LIN {X 0,Y 504.364,Z 1241.928,A -85,B 0,C 180,E1 24651.564,E2 24651.564} C_VEL
LIN {X 0,Y 504.744,Z 1235.291,A -85,B 0,C 180,E1 24649.268,E2 24649.268} C_VEL
LIN {X 0,Y 505.368,Z 1226.948,A -85,B 0,C 180,E1 24646.965,E2 24646.965} C_VEL
LIN {X 0,Y 506.263,Z 1217.284,A -85,B 0,C 180,E1 24644.771,E2 24644.771} C_VEL
LIN {X 0,Y 507.475,Z 1205.57,A -85,B 0,C 180,E1 24642.573,E2 24642.573} C_VEL
LIN {X 0,Y 508.891,Z 1193.016,A -85,B 0,C 180,E1 24640.585,E2 24640.585} C_VEL
LIN {X 0,Y 510.606,Z 1178.677,A -85,B 0,C 180,E1 24638.639,E2 24638.639} C_VEL
LIN {X 0,Y 512.557,Z 1162.738,A -85,B 0,C 180,E1 24636.793,E2 24636.793} C_VEL
LIN {X 0,Y 514.559,Z 1146.108,A -85,B 0,C 180,E1 24635.16,E2 24635.16} C_VEL
LIN {X 0,Y 516.658,Z 1128.097,A -85,B 0,C 180,E1 24633.644,E2 24633.644} C_VEL
LIN {X 0,Y 518.812,Z 1108.718,A -85,B 0,C 180,E1 24632.261,E2 24632.261} C_VEL
LIN {X 0,Y 520.852,Z 1088.73,A -85,B 0,C 180,E1 24631.068,E2 24631.068} C_VEL
LIN {X 0,Y 522.71,Z 1067.81,A -85,B 0,C 180,E1 24630.048,E2 24630.048} C_VEL
LIN {X 0,Y 524.415,Z 1045.644,A -85,B 0,C 180,E1 24629.185,E2 24629.185} C_VEL
LIN {X 0,Y 525.788,Z 1023.231,A -85,B 0,C 180,E1 24628.517,E2 24628.517} C_VEL
LIN {X 0,Y 526.855,Z 1000.213,A -85,B 0,C 180,E1 24628.032,E2 24628.032} C_VEL
LIN {X 0,Y 534.144,Z 792.221,A -85,B 0,C 180,E1 24624.636,E2 24624.636} C_VEL
LIN {X 0,Y 535.779,Z 746.404,A -85,B 0,C 180,E1 24623.864,E2 24623.864} C_VEL
LIN {X 0,Y 532.938,Z 733.68,A -85,B 0,C 180,E1 24623.419,E2 24623.419} C_VEL
LIN {X 0,Y 518.726,Z 705.757,A -85,B 0,C 180,E1 24621.804,E2 24621.804} C_VEL
LIN {X 0,Y 511.196,Z 684.324,A -85,B 0,C 180,E1 24619.027,E2 24619.027} C_VEL
LIN {X 0,Y 505.862,Z 669.652,A -85,B 0,C 180,E1 24617.044,E2 24617.044} C_VEL
LIN {X 0,Y 505.876,Z 669.66,A -85,B 0,C 180,E1 24613.461,E2 24613.461} C_VEL
LIN {X 0,Y 505.86,Z 669.653,A -85,B 0,C 180,E1 24609.921,E2 24609.921} C_VEL
LIN {X 0,Y 505.869,Z 669.652,A -85,B 0,C 180,E1 24606.369,E2 24606.369} C_VEL
LIN {X 0,Y 505.872,Z 669.655,A -85,B 0,C 180,E1 24602.792,E2 24602.792} C_VEL
LIN {X 0,Y 505.863,Z 669.654,A -85,B 0,C 180,E1 24599.345,E2 24599.345} C_VEL
LIN {X 0,Y 505.866,Z 669.654,A -85,B 0,C 180,E1 24595.777,E2 24595.777} C_VEL
LIN {X 0,Y 505.86,Z 669.657,A -85,B 0,C 180,E1 24592.305,E2 24592.305} C_VEL
LIN {X 0,Y 505.871,Z 669.651,A -85,B 0,C 180,E1 24588.776,E2 24588.776} C_VEL
LIN {X 0,Y 505.866,Z 669.656,A -85,B 0,C 180,E1 24588.016,E2 24588.016} C_VEL
LIN {X 0,Y 504.876,Z 669.777,A -85,B 0,C 180,E1 24587.144,E2 24587.144} C_VEL
LIN {X 0,Y 498.35,Z 670.589,A -85,B 0,C 180,E1 24584.628,E2 24584.628} C_VEL
LIN {X 0,Y 497.917,Z 670.638,A -85,B 0,C 180,E1 24584.052,E2 24584.052} C_VEL
LIN {X 0,Y 497.931,Z 670.642,A -85,B 0,C 180,E1 24580.531,E2 24580.531} C_VEL
LIN {X 0,Y 497.921,Z 670.643,A -85,B 0,C 180,E1 24576.922,E2 24576.922} C_VEL
LIN {X 0,Y 497.921,Z 670.639,A -85,B 0,C 180,E1 24573.34,E2 24573.34} C_VEL
LIN {X 0,Y 497.923,Z 670.634,A -85,B 0,C 180,E1 24569.771,E2 24569.771} C_VEL
LIN {X 0,Y 497.917,Z 670.635,A -85,B 0,C 180,E1 24566.317,E2 24566.317} C_VEL
LIN {X 0,Y 497.936,Z 670.635,A -85,B 0,C 180,E1 24562.734,E2 24562.734} C_VEL
LIN {X 0,Y 497.917,Z 670.636,A -85,B 0,C 180,E1 24559.109,E2 24559.109} C_VEL
LIN {X 0,Y 497.936,Z 670.637,A -85,B 0,C 180,E1 24555.583,E2 24555.583} C_VEL
LIN {X 0,Y 497.923,Z 670.645,A -85,B 0,C 180,E1 24551.988,E2 24551.988} C_VEL
LIN {X 0,Y 497.926,Z 670.645,A -85,B 0,C 180,E1 24548.397,E2 24548.397} C_VEL
LIN {X 0,Y 497.925,Z 670.639,A -85,B 0,C 180,E1 24544.806,E2 24544.806} C_VEL
LIN {X 0,Y 497.922,Z 670.645,A -85,B 0,C 180,E1 24541.321,E2 24541.321} C_VEL
LIN {X 0,Y 497.925,Z 670.626,A -85,B 0,C 180,E1 24537.852,E2 24537.852} C_VEL
LIN {X 0,Y 497.919,Z 670.631,A -85,B 0,C 180,E1 24534.244,E2 24534.244} C_VEL
LIN {X 0,Y 497.955,Z 670.843,A -85,B 0,C 180,E1 24533.437,E2 24533.437} C_VEL
LIN {X 0,Y 506.765,Z 692.841,A -85,B 0,C 180,E1 24530.265,E2 24530.265} C_VEL
LIN {X 0,Y 514.424,Z 713.346,A -85,B 0,C 180,E1 24527.515,E2 24527.515} C_VEL
LIN {X 0,Y 521.93,Z 735.394,A -85,B 0,C 180,E1 24524.785,E2 24524.785} C_VEL
LIN {X 0,Y 522.331,Z 737.49,A -85,B 0,C 180,E1 24524.555,E2 24524.555} C_VEL
LIN {X 0,Y 518.753,Z 774.196,A -85,B 0,C 180,E1 24521.386,E2 24521.386} C_VEL
LIN {X 0,Y 514.969,Z 815.795,A -85,B 0,C 180,E1 24517.848,E2 24517.848} C_VEL
LIN {X 0,Y 511.442,Z 859.058,A -85,B 0,C 180,E1 24514.214,E2 24514.214} C_VEL
LIN {X 0,Y 508.148,Z 905.295,A -85,B 0,C 180,E1 24510.378,E2 24510.378} C_VEL
LIN {X 0,Y 507.992,Z 908.898,A -85,B 0,C 180,E1 24510.113,E2 24510.113} C_VEL
LIN {X 0,Y 508.886,Z 919.664,A -85,B 0,C 180,E1 24509.842,E2 24509.842} C_VEL
LIN {X 0,Y 504.35,Z 1050.728,A -85,B 0,C 180,E1 24507.128,E2 24507.128} C_VEL
LIN {X 0,Y 503.904,Z 1067.841,A -85,B 0,C 180,E1 24506.613,E2 24506.613} C_VEL
LIN {X 0,Y 503.25,Z 1083.698,A -85,B 0,C 180,E1 24505.92,E2 24505.92} C_VEL
LIN {X 0,Y 502.43,Z 1099.334,A -85,B 0,C 180,E1 24505.017,E2 24505.017} C_VEL
LIN {X 0,Y 501.517,Z 1113.85,A -85,B 0,C 180,E1 24503.937,E2 24503.937} C_VEL
LIN {X 0,Y 500.596,Z 1127.537,A -85,B 0,C 180,E1 24502.668,E2 24502.668} C_VEL
LIN {X 0,Y 499.652,Z 1140.382,A -85,B 0,C 180,E1 24501.172,E2 24501.172} C_VEL
LIN {X 0,Y 498.883,Z 1150.749,A -85,B 0,C 180,E1 24499.677,E2 24499.677} C_VEL
LIN {X 0,Y 498.188,Z 1160.6,A -85,B 0,C 180,E1 24497.883,E2 24497.883} C_VEL
LIN {X 0,Y 497.736,Z 1167.748,A -85,B 0,C 180,E1 24496.215,E2 24496.215} C_VEL
LIN {X 0,Y 497.42,Z 1173.818,A -85,B 0,C 180,E1 24494.315,E2 24494.315} C_VEL
LIN {X 0,Y 497.291,Z 1177.76,A -85,B 0,C 180,E1 24492.542,E2 24492.542} C_VEL
LIN {X 0,Y 497.285,Z 1180.289,A -85,B 0,C 180,E1 24490.521,E2 24490.521} C_VEL
LIN {X 0,Y 497.431,Z 1180.907,A -85,B 0,C 180,E1 24488.671,E2 24488.671} C_VEL
LIN {X 0,Y 497.725,Z 1179.692,A -85,B 0,C 180,E1 24486.691,E2 24486.691} C_VEL
LIN {X 0,Y 498.203,Z 1176.854,A -85,B 0,C 180,E1 24484.835,E2 24484.835} C_VEL
LIN {X 0,Y 498.95,Z 1171.888,A -85,B 0,C 180,E1 24482.872,E2 24482.872} C_VEL
LIN {X 0,Y 499.852,Z 1165.769,A -85,B 0,C 180,E1 24481.146,E2 24481.146} C_VEL
LIN {X 0,Y 501.108,Z 1157.14,A -85,B 0,C 180,E1 24479.314,E2 24479.314} C_VEL
LIN {X 0,Y 502.459,Z 1147.46,A -85,B 0,C 180,E1 24477.719,E2 24477.719} C_VEL
LIN {X 0,Y 503.927,Z 1136.358,A -85,B 0,C 180,E1 24476.246,E2 24476.246} C_VEL
LIN {X 0,Y 505.458,Z 1123.633,A -85,B 0,C 180,E1 24474.893,E2 24474.893} C_VEL
LIN {X 0,Y 506.866,Z 1110.62,A -85,B 0,C 180,E1 24473.771,E2 24473.771} C_VEL
LIN {X 0,Y 508.237,Z 1095.771,A -85,B 0,C 180,E1 24472.767,E2 24472.767} C_VEL
LIN {X 0,Y 509.323,Z 1081.041,A -85,B 0,C 180,E1 24471.988,E2 24471.988} C_VEL
LIN {X 0,Y 510.261,Z 1063.639,A -85,B 0,C 180,E1 24471.307,E2 24471.307} C_VEL
LIN {X 0,Y 513.071,Z 1023.611,A -85,B 0,C 180,E1 24470.111,E2 24470.111} C_VEL
LIN {X 0,Y 519.657,Z 948.637,A -85,B 0,C 180,E1 24468.048,E2 24468.048} C_VEL
LIN {X 0,Y 521.331,Z 927.047,A -85,B 0,C 180,E1 24467.49,E2 24467.49} C_VEL
LIN {X 0,Y 528.249,Z 885.776,A -85,B 0,C 180,E1 24463.562,E2 24463.562} C_VEL
LIN {X 0,Y 536.223,Z 847.729,A -85,B 0,C 180,E1 24459.82,E2 24459.82} C_VEL
LIN {X 0,Y 545.73,Z 811.629,A -85,B 0,C 180,E1 24456.114,E2 24456.114} C_VEL
LIN {X 0,Y 554.554,Z 784.609,A -85,B 0,C 180,E1 24453.207,E2 24453.207} C_VEL
LIN {X 0,Y 556.027,Z 780.377,A -85,B 0,C 180,E1 24452.706,E2 24452.706} C_VEL
LIN {X 0,Y 555.302,Z 773.817,A -85,B 0,C 180,E1 24450.793,E2 24450.793} C_VEL
LIN {X 0,Y 554.864,Z 769.209,A -85,B 0,C 180,E1 24448.856,E2 24448.856} C_VEL
LIN {X 0,Y 554.855,Z 767.416,A -85,B 0,C 180,E1 24447.686,E2 24447.686} C_VEL
LIN {X 0,Y 555.608,Z 765.75,A -85,B 0,C 180,E1 24445.507,E2 24445.507} C_VEL
LIN {X 0,Y 555.776,Z 766.406,A -85,B 0,C 180,E1 24444.582,E2 24444.582} C_VEL
LIN {X 0,Y 556.536,Z 769.26,A -85,B 0,C 180,E1 24442.737,E2 24442.737} C_VEL
LIN {X 0,Y 557.449,Z 773.099,A -85,B 0,C 180,E1 24441.301,E2 24441.301} C_VEL
LIN {X 0,Y 547.171,Z 799.995,A -85,B 0,C 180,E1 24438.917,E2 24438.917} C_VEL
LIN {X 0,Y 539.997,Z 825.145,A -85,B 0,C 180,E1 24436.691,E2 24436.691} C_VEL
LIN {X 0,Y 536.29,Z 846.795,A -85,B 0,C 180,E1 24434.657,E2 24434.657} C_VEL
LIN {X 0,Y 535.325,Z 864.261,A -85,B 0,C 180,E1 24432.93,E2 24432.93} C_VEL
LIN {X 0,Y 536.577,Z 881.954,A -85,B 0,C 180,E1 24431.082,E2 24431.082} C_VEL
LIN {X 0,Y 540.082,Z 898.355,A -85,B 0,C 180,E1 24429.297,E2 24429.297} C_VEL
LIN {X 0,Y 545.937,Z 914.131,A -85,B 0,C 180,E1 24427.529,E2 24427.529} C_VEL
LIN {X 0,Y 553.358,Z 927.813,A -85,B 0,C 180,E1 24425.951,E2 24425.951} C_VEL
LIN {X 0,Y 553.874,Z 928.862,A -85,B 0,C 180,E1 24425.839,E2 24425.839} C_VEL
LIN {X 0,Y 543.51,Z 949.382,A -85,B 0,C 180,E1 24425.09,E2 24425.09} C_VEL
LIN {X 0,Y 530.676,Z 977.187,A -85,B 0,C 180,E1 24423.961,E2 24423.961} C_VEL
LIN {X 0,Y 521.338,Z 1002.518,A -85,B 0,C 180,E1 24422.778,E2 24422.778} C_VEL
LIN {X 0,Y 518.892,Z 1027.417,A -85,B 0,C 180,E1 24422.456,E2 24422.456} C_VEL
LIN {X 0,Y 517.522,Z 1062.325,A -85,B 0,C 180,E1 24421.831,E2 24421.831} C_VEL
LIN {X 0,Y 516.081,Z 1085.156,A -85,B 0,C 180,E1 24421.23,E2 24421.23} C_VEL
LIN {X 0,Y 514.305,Z 1107.549,A -85,B 0,C 180,E1 24420.426,E2 24420.426} C_VEL
LIN {X 0,Y 512.324,Z 1128.678,A -85,B 0,C 180,E1 24419.458,E2 24419.458} C_VEL
LIN {X 0,Y 510.136,Z 1150.077,A -85,B 0,C 180,E1 24418.25,E2 24418.25} C_VEL
LIN {X 0,Y 507.97,Z 1169.722,A -85,B 0,C 180,E1 24416.913,E2 24416.913} C_VEL
LIN {X 0,Y 505.782,Z 1188.665,A -85,B 0,C 180,E1 24415.384,E2 24415.384} C_VEL
LIN {X 0,Y 503.683,Z 1206.377,A -85,B 0,C 180,E1 24413.684,E2 24413.684} C_VEL
LIN {X 0,Y 501.781,Z 1222.458,A -85,B 0,C 180,E1 24411.876,E2 24411.876} C_VEL
LIN {X 0,Y 500.177,Z 1236.908,A -85,B 0,C 180,E1 24409.987,E2 24409.987} C_VEL
LIN {X 0,Y 498.742,Z 1250.762,A -85,B 0,C 180,E1 24407.861,E2 24407.861} C_VEL
LIN {X 0,Y 497.682,Z 1262.373,A -85,B 0,C 180,E1 24405.735,E2 24405.735} C_VEL
LIN {X 0,Y 496.884,Z 1273.169,A -85,B 0,C 180,E1 24403.379,E2 24403.379} C_VEL
LIN {X 0,Y 496.419,Z 1281.59,A -85,B 0,C 180,E1 24401.147,E2 24401.147} C_VEL
LIN {X 0,Y 496.194,Z 1288.215,A -85,B 0,C 180,E1 24398.925,E2 24398.925} C_VEL
LIN {X 0,Y 496.115,Z 1293.775,A -85,B 0,C 180,E1 24396.477,E2 24396.477} C_VEL
LIN {X 0,Y 496.133,Z 1297.446,A -85,B 0,C 180,E1 24394.159,E2 24394.159} C_VEL
LIN {X 0,Y 496.171,Z 1299.407,A -85,B 0,C 180,E1 24391.846,E2 24391.846} C_VEL
LIN {X 0,Y 496.179,Z 1299.871,A -85,B 0,C 180,E1 24389.421,E2 24389.421} C_VEL
LIN {X 0,Y 496.163,Z 1298.798,A -85,B 0,C 180,E1 24387.226,E2 24387.226} C_VEL
LIN {X 0,Y 496.121,Z 1295.944,A -85,B 0,C 180,E1 24384.795,E2 24384.795} C_VEL
LIN {X 0,Y 496.145,Z 1291.669,A -85,B 0,C 180,E1 24382.471,E2 24382.471} C_VEL
LIN {X 0,Y 496.271,Z 1285.615,A -85,B 0,C 180,E1 24380.138,E2 24380.138} C_VEL
LIN {X 0,Y 496.616,Z 1277.824,A -85,B 0,C 180,E1 24377.794,E2 24377.794} C_VEL
LIN {X 0,Y 497.2,Z 1268.724,A -85,B 0,C 180,E1 24375.558,E2 24375.558} C_VEL
LIN {X 0,Y 498.121,Z 1257.595,A -85,B 0,C 180,E1 24373.317,E2 24373.317} C_VEL
LIN {X 0,Y 499.351,Z 1245.086,A -85,B 0,C 180,E1 24371.192,E2 24371.192} C_VEL
LIN {X 0,Y 500.876,Z 1231.302,A -85,B 0,C 180,E1 24369.185,E2 24369.185} C_VEL
LIN {X 0,Y 502.803,Z 1215.123,A -85,B 0,C 180,E1 24367.182,E2 24367.182} C_VEL
LIN {X 0,Y 504.856,Z 1198.42,A -85,B 0,C 180,E1 24365.422,E2 24365.422} C_VEL
LIN {X 0,Y 507.196,Z 1179.761,A -85,B 0,C 180,E1 24363.736,E2 24363.736} C_VEL
LIN {X 0,Y 509.611,Z 1160.303,A -85,B 0,C 180,E1 24362.239,E2 24362.239} C_VEL
LIN {X 0,Y 512.103,Z 1139.839,A -85,B 0,C 180,E1 24360.909,E2 24360.909} C_VEL
LIN {X 0,Y 514.507,Z 1118.825,A -85,B 0,C 180,E1 24359.778,E2 24359.778} C_VEL
LIN {X 0,Y 516.923,Z 1096.126,A -85,B 0,C 180,E1 24358.774,E2 24358.774} C_VEL
LIN {X 0,Y 519.31,Z 1071.964,A -85,B 0,C 180,E1 24357.938,E2 24357.938} C_VEL
LIN {X 0,Y 521.333,Z 1047.272,A -85,B 0,C 180,E1 24357.297,E2 24357.297} C_VEL
LIN {X 0,Y 523.291,Z 1020.268,A -85,B 0,C 180,E1 24356.763,E2 24356.763} C_VEL
LIN {X 0,Y 526.834,Z 993.87,A -85,B 0,C 180,E1 24356.393,E2 24356.393} C_VEL
LIN {X 0,Y 528.818,Z 981.657,A -85,B 0,C 180,E1 24356.226,E2 24356.226} C_VEL
LIN {X 0,Y 537.469,Z 962.627,A -85,B 0,C 180,E1 24355.364,E2 24355.364} C_VEL
LIN {X 0,Y 551.978,Z 933.996,A -85,B 0,C 180,E1 24354.189,E2 24354.189} C_VEL
LIN {X 0,Y 554.447,Z 929.286,A -85,B 0,C 180,E1 24354.006,E2 24354.006} C_VEL
LIN {X 0,Y 545.465,Z 913.489,A -85,B 0,C 180,E1 24352.45,E2 24352.45} C_VEL
LIN {X 0,Y 538.162,Z 895.688,A -85,B 0,C 180,E1 24350.785,E2 24350.785} C_VEL
LIN {X 0,Y 533.179,Z 877.53,A -85,B 0,C 180,E1 24349.174,E2 24349.174} C_VEL
LIN {X 0,Y 529.999,Z 856.994,A -85,B 0,C 180,E1 24347.453,E2 24347.453} C_VEL
LIN {X 0,Y 529.011,Z 834.745,A -85,B 0,C 180,E1 24345.708,E2 24345.708} C_VEL
LIN {X 0,Y 530.151,Z 810.275,A -85,B 0,C 180,E1 24343.906,E2 24343.906} C_VEL
LIN {X 0,Y 534.248,Z 775.142,A -85,B 0,C 180,E1 24341.454,E2 24341.454} C_VEL
LIN {X 0,Y 537.68,Z 769.168,A -85,B 0,C 180,E1 24340.728,E2 24340.728} C_VEL
LIN {X 0,Y 542.857,Z 759.339,A -85,B 0,C 180,E1 24339.9,E2 24339.9} C_VEL
LIN {X 0,Y 545.665,Z 757.3,A -85,B 0,C 180,E1 24339.308,E2 24339.308} C_VEL
LIN {X 0,Y 549.092,Z 755.477,A -85,B 0,C 180,E1 24338.634,E2 24338.634} C_VEL
LIN {X 0,Y 538.742,Z 835.57,A -85,B 0,C 180,E1 24336.721,E2 24336.721} C_VEL
LIN {X 0,Y 530.844,Z 913.19,A -85,B 0,C 180,E1 24334.924,E2 24334.924} C_VEL
LIN {X 0,Y 525.076,Z 987.708,A -85,B 0,C 180,E1 24333.314,E2 24333.314} C_VEL
LIN {X 0,Y 522.716,Z 1023.697,A -85,B 0,C 180,E1 24332.523,E2 24332.523} C_VEL
LIN {X 0,Y 520.89,Z 1047.072,A -85,B 0,C 180,E1 24331.798,E2 24331.798} C_VEL
LIN {X 0,Y 518.661,Z 1070.49,A -85,B 0,C 180,E1 24330.851,E2 24330.851} C_VEL
LIN {X 0,Y 516.264,Z 1092.595,A -85,B 0,C 180,E1 24329.724,E2 24329.724} C_VEL
LIN {X 0,Y 513.818,Z 1112.739,A -85,B 0,C 180,E1 24328.475,E2 24328.475} C_VEL
LIN {X 0,Y 511.287,Z 1132.087,A -85,B 0,C 180,E1 24327.045,E2 24327.045} C_VEL
LIN {X 0,Y 508.747,Z 1150.526,A -85,B 0,C 180,E1 24325.432,E2 24325.432} C_VEL
LIN {X 0,Y 506.333,Z 1167.423,A -85,B 0,C 180,E1 24323.695,E2 24323.695} C_VEL
LIN {X 0,Y 504.035,Z 1183.242,A -85,B 0,C 180,E1 24321.775,E2 24321.775} C_VEL
LIN {X 0,Y 502.033,Z 1197.078,A -85,B 0,C 180,E1 24319.791,E2 24319.791} C_VEL
LIN {X 0,Y 500.215,Z 1210.203,A -85,B 0,C 180,E1 24317.568,E2 24317.568} C_VEL
LIN {X 0,Y 498.815,Z 1221.199,A -85,B 0,C 180,E1 24315.343,E2 24315.343} C_VEL
LIN {X 0,Y 497.729,Z 1230.767,A -85,B 0,C 180,E1 24313.003,E2 24313.003} C_VEL
LIN {X 0,Y 496.982,Z 1238.369,A -85,B 0,C 180,E1 24310.667,E2 24310.667} C_VEL
LIN {X 0,Y 496.49,Z 1244.569,A -85,B 0,C 180,E1 24308.221,E2 24308.221} C_VEL
LIN {X 0,Y 496.231,Z 1249.071,A -85,B 0,C 180,E1 24305.782,E2 24305.782} C_VEL
LIN {X 0,Y 496.096,Z 1251.736,A -85,B 0,C 180,E1 24303.467,E2 24303.467} C_VEL
LIN {X 0,Y 496.049,Z 1252.986,A -85,B 0,C 180,E1 24301.039,E2 24301.039} C_VEL
LIN {X 0,Y 496.034,Z 1252.746,A -85,B 0,C 180,E1 24298.729,E2 24298.729} C_VEL
LIN {X 0,Y 496.057,Z 1250.806,A -85,B 0,C 180,E1 24296.302,E2 24296.302} C_VEL
LIN {X 0,Y 496.163,Z 1247.071,A -85,B 0,C 180,E1 24293.752,E2 24293.752} C_VEL
LIN {X 0,Y 496.395,Z 1242.114,A -85,B 0,C 180,E1 24291.428,E2 24291.428} C_VEL
LIN {X 0,Y 496.825,Z 1235.048,A -85,B 0,C 180,E1 24288.978,E2 24288.978} C_VEL
LIN {X 0,Y 497.503,Z 1226.494,A -85,B 0,C 180,E1 24286.636,E2 24286.636} C_VEL
LIN {X 0,Y 498.519,Z 1216.007,A -85,B 0,C 180,E1 24284.29,E2 24284.29} C_VEL
LIN {X 0,Y 499.765,Z 1204.724,A -85,B 0,C 180,E1 24282.175,E2 24282.175} C_VEL
LIN {X 0,Y 501.347,Z 1191.247,A -85,B 0,C 180,E1 24280.059,E2 24280.059} C_VEL
LIN {X 0,Y 503.206,Z 1176.294,A -85,B 0,C 180,E1 24278.064,E2 24278.064} C_VEL
LIN {X 0,Y 505.279,Z 1159.817,A -85,B 0,C 180,E1 24276.191,E2 24276.191} C_VEL
LIN {X 0,Y 507.389,Z 1143.021,A -85,B 0,C 180,E1 24274.557,E2 24274.557} C_VEL
LIN {X 0,Y 509.666,Z 1123.886,A -85,B 0,C 180,E1 24272.988,E2 24272.988} C_VEL
LIN {X 0,Y 511.803,Z 1104.612,A -85,B 0,C 180,E1 24271.657,E2 24271.657} C_VEL
LIN {X 0,Y 513.956,Z 1083.523,A -85,B 0,C 180,E1 24270.444,E2 24270.444} C_VEL
LIN {X 0,Y 515.867,Z 1062.333,A -85,B 0,C 180,E1 24269.448,E2 24269.448} C_VEL
LIN {X 0,Y 517.522,Z 1040.269,A -85,B 0,C 180,E1 24268.627,E2 24268.627} C_VEL
LIN {X 0,Y 518.851,Z 1017.754,A -85,B 0,C 180,E1 24268.005,E2 24268.005} C_VEL
LIN {X 0,Y 519.95,Z 991.242,A -85,B 0,C 180,E1 24267.501,E2 24267.501} C_VEL
LIN {X 0,Y 527.629,Z 784.848,A -85,B 0,C 180,E1 24264.06,E2 24264.06} C_VEL
LIN {X 0,Y 529.017,Z 747.99,A -85,B 0,C 180,E1 24263.424,E2 24263.424} C_VEL
LIN {X 0,Y 526.552,Z 737.144,A -85,B 0,C 180,E1 24263.034,E2 24263.034} C_VEL
LIN {X 0,Y 510.662,Z 706.055,A -85,B 0,C 180,E1 24261.197,E2 24261.197} C_VEL
LIN {X 0,Y 503.381,Z 685.505,A -85,B 0,C 180,E1 24258.492,E2 24258.492} C_VEL
LIN {X 0,Y 497.922,Z 670.642,A -85,B 0,C 180,E1 24256.465,E2 24256.465} C_VEL
LIN {X 0,Y 497.927,Z 670.642,A -85,B 0,C 180,E1 24252.903,E2 24252.903} C_VEL
LIN {X 0,Y 497.927,Z 670.644,A -85,B 0,C 180,E1 24249.365,E2 24249.365} C_VEL
LIN {X 0,Y 497.935,Z 670.647,A -85,B 0,C 180,E1 24245.78,E2 24245.78} C_VEL
LIN {X 0,Y 497.929,Z 670.643,A -85,B 0,C 180,E1 24242.152,E2 24242.152} C_VEL
LIN {X 0,Y 497.922,Z 670.644,A -85,B 0,C 180,E1 24238.651,E2 24238.651} C_VEL
LIN {X 0,Y 497.936,Z 670.645,A -85,B 0,C 180,E1 24235.07,E2 24235.07} C_VEL
LIN {X 0,Y 497.923,Z 670.645,A -85,B 0,C 180,E1 24231.562,E2 24231.562} C_VEL
LIN {X 0,Y 497.928,Z 670.645,A -85,B 0,C 180,E1 24228.015,E2 24228.015} C_VEL
LIN {X 0,Y 497.928,Z 670.639,A -85,B 0,C 180,E1 24224.42,E2 24224.42} C_VEL
LIN {X 0,Y 497.917,Z 670.638,A -85,B 0,C 180,E1 24224.052,E2 24224.052} C_VEL
LIN {X 0,Y 496.935,Z 670.759,A -85,B 0,C 180,E1 24223.166,E2 24223.166} C_VEL
LIN {X 0,Y 490.419,Z 671.58,A -85,B 0,C 180,E1 24220.609,E2 24220.609} C_VEL
LIN {X 0,Y 489.982,Z 671.632,A -85,B 0,C 180,E1 24220.024,E2 24220.024} C_VEL
LIN {X 0,Y 489.988,Z 671.631,A -85,B 0,C 180,E1 24216.446,E2 24216.446} C_VEL
LIN {X 0,Y 489.98,Z 671.629,A -85,B 0,C 180,E1 24212.809,E2 24212.809} C_VEL
LIN {X 0,Y 489.98,Z 671.624,A -85,B 0,C 180,E1 24209.3,E2 24209.3} C_VEL
LIN {X 0,Y 489.991,Z 671.622,A -85,B 0,C 180,E1 24205.672,E2 24205.672} C_VEL
LIN {X 0,Y 489.978,Z 671.625,A -85,B 0,C 180,E1 24202.143,E2 24202.143} C_VEL
LIN {X 0,Y 489.986,Z 671.624,A -85,B 0,C 180,E1 24198.585,E2 24198.585} C_VEL
LIN {X 0,Y 489.983,Z 671.63,A -85,B 0,C 180,E1 24194.981,E2 24194.981} C_VEL
LIN {X 0,Y 489.988,Z 671.634,A -85,B 0,C 180,E1 24191.439,E2 24191.439} C_VEL
LIN {X 0,Y 489.983,Z 671.634,A -85,B 0,C 180,E1 24187.822,E2 24187.822} C_VEL
LIN {X 0,Y 489.984,Z 671.631,A -85,B 0,C 180,E1 24184.239,E2 24184.239} C_VEL
LIN {X 0,Y 489.997,Z 671.63,A -85,B 0,C 180,E1 24180.544,E2 24180.544} C_VEL
LIN {X 0,Y 489.983,Z 671.618,A -85,B 0,C 180,E1 24176.988,E2 24176.988} C_VEL
LIN {X 0,Y 490.011,Z 671.847,A -85,B 0,C 180,E1 24174.155,E2 24174.155} C_VEL
LIN {X 0,Y 498.364,Z 692.439,A -85,B 0,C 180,E1 24171.101,E2 24171.101} C_VEL
LIN {X 0,Y 506.167,Z 713.033,A -85,B 0,C 180,E1 24168.266,E2 24168.266} C_VEL
LIN {X 0,Y 513.881,Z 735.453,A -85,B 0,C 180,E1 24165.41,E2 24165.41} C_VEL
LIN {X 0,Y 515.236,Z 740.019,A -85,B 0,C 180,E1 24164.864,E2 24164.864} C_VEL
LIN {X 0,Y 511.531,Z 776.997,A -85,B 0,C 180,E1 24161.652,E2 24161.652} C_VEL
LIN {X 0,Y 507.592,Z 818.716,A -85,B 0,C 180,E1 24158.066,E2 24158.066} C_VEL
LIN {X 0,Y 503.893,Z 862.26,A -85,B 0,C 180,E1 24154.367,E2 24154.367} C_VEL
LIN {X 0,Y 500.56,Z 907.377,A -85,B 0,C 180,E1 24150.582,E2 24150.582} C_VEL
LIN {X 0,Y 500.515,Z 909.781,A -85,B 0,C 180,E1 24150.426,E2 24150.426} C_VEL
LIN {X 0,Y 501.381,Z 920.588,A -85,B 0,C 180,E1 24150.149,E2 24150.149} C_VEL
LIN {X 0,Y 496.68,Z 1050.301,A -85,B 0,C 180,E1 24147.399,E2 24147.399} C_VEL
LIN {X 0,Y 496.206,Z 1067.96,A -85,B 0,C 180,E1 24146.865,E2 24146.865} C_VEL
LIN {X 0,Y 495.524,Z 1084.054,A -85,B 0,C 180,E1 24146.155,E2 24146.155} C_VEL
LIN {X 0,Y 494.678,Z 1099.617,A -85,B 0,C 180,E1 24145.245,E2 24145.245} C_VEL
LIN {X 0,Y 493.731,Z 1114.23,A -85,B 0,C 180,E1 24144.148,E2 24144.148} C_VEL
LIN {X 0,Y 492.81,Z 1127.454,A -85,B 0,C 180,E1 24142.912,E2 24142.912} C_VEL
LIN {X 0,Y 491.942,Z 1139,A -85,B 0,C 180,E1 24141.586,E2 24141.586} C_VEL
LIN {X 0,Y 491.08,Z 1150.184,A -85,B 0,C 180,E1 24140.003,E2 24140.003} C_VEL
LIN {X 0,Y 490.414,Z 1159.187,A -85,B 0,C 180,E1 24138.423,E2 24138.423} C_VEL
LIN {X 0,Y 489.876,Z 1167.32,A -85,B 0,C 180,E1 24136.604,E2 24136.604} C_VEL
LIN {X 0,Y 489.53,Z 1173.484,A -85,B 0,C 180,E1 24134.793,E2 24134.793} C_VEL
LIN {X 0,Y 489.348,Z 1178.3,A -85,B 0,C 180,E1 24132.749,E2 24132.749} C_VEL
LIN {X 0,Y 489.332,Z 1180.969,A -85,B 0,C 180,E1 24130.836,E2 24130.836} C_VEL
LIN {X 0,Y 489.477,Z 1181.921,A -85,B 0,C 180,E1 24128.813,E2 24128.813} C_VEL
LIN {X 0,Y 489.762,Z 1181.073,A -85,B 0,C 180,E1 24126.918,E2 24126.918} C_VEL
LIN {X 0,Y 490.271,Z 1178.356,A -85,B 0,C 180,E1 24124.914,E2 24124.914} C_VEL
LIN {X 0,Y 490.992,Z 1174.008,A -85,B 0,C 180,E1 24123.035,E2 24123.035} C_VEL
LIN {X 0,Y 492.016,Z 1167.604,A -85,B 0,C 180,E1 24121.108,E2 24121.108} C_VEL
LIN {X 0,Y 493.269,Z 1159.489,A -85,B 0,C 180,E1 24119.303,E2 24119.303} C_VEL
LIN {X 0,Y 494.684,Z 1150.259,A -85,B 0,C 180,E1 24117.683,E2 24117.683} C_VEL
LIN {X 0,Y 496.323,Z 1138.65,A -85,B 0,C 180,E1 24116.072,E2 24116.072} C_VEL
LIN {X 0,Y 497.864,Z 1126.874,A -85,B 0,C 180,E1 24114.757,E2 24114.757} C_VEL
LIN {X 0,Y 499.469,Z 1112.928,A -85,B 0,C 180,E1 24113.505,E2 24113.505} C_VEL
LIN {X 0,Y 500.92,Z 1098.61,A -85,B 0,C 180,E1 24112.487,E2 24112.487} C_VEL
LIN {X 0,Y 502.179,Z 1083.506,A -85,B 0,C 180,E1 24111.642,E2 24111.642} C_VEL
LIN {X 0,Y 503.162,Z 1066.735,A -85,B 0,C 180,E1 24110.953,E2 24110.953} C_VEL
LIN {X 0,Y 505.892,Z 1029.39,A -85,B 0,C 180,E1 24109.779,E2 24109.779} C_VEL
LIN {X 0,Y 512.761,Z 955.756,A -85,B 0,C 180,E1 24107.677,E2 24107.677} C_VEL
LIN {X 0,Y 515.019,Z 928.622,A -85,B 0,C 180,E1 24106.96,E2 24106.96} C_VEL
LIN {X 0,Y 522.253,Z 887.889,A -85,B 0,C 180,E1 24103.024,E2 24103.024} C_VEL
LIN {X 0,Y 530.696,Z 850.247,A -85,B 0,C 180,E1 24099.255,E2 24099.255} C_VEL
LIN {X 0,Y 540.105,Z 816.488,A -85,B 0,C 180,E1 24095.733,E2 24095.733} C_VEL
LIN {X 0,Y 549.352,Z 789.709,A -85,B 0,C 180,E1 24092.816,E2 24092.816} C_VEL
LIN {X 0,Y 550.844,Z 785.492,A -85,B 0,C 180,E1 24092.31,E2 24092.31} C_VEL
LIN {X 0,Y 550.394,Z 779.565,A -85,B 0,C 180,E1 24090.476,E2 24090.476} C_VEL
LIN {X 0,Y 550.194,Z 775.471,A -85,B 0,C 180,E1 24088.662,E2 24088.662} C_VEL
LIN {X 0,Y 550.251,Z 773.894,A -85,B 0,C 180,E1 24087.584,E2 24087.584} C_VEL
LIN {X 0,Y 551.076,Z 772.341,A -85,B 0,C 180,E1 24085.458,E2 24085.458} C_VEL
LIN {X 0,Y 551.221,Z 773.117,A -85,B 0,C 180,E1 24084.516,E2 24084.516} C_VEL
LIN {X 0,Y 551.914,Z 775.887,A -85,B 0,C 180,E1 24082.764,E2 24082.764} C_VEL
LIN {X 0,Y 552.46,Z 778.589,A -85,B 0,C 180,E1 24081.725,E2 24081.725} C_VEL
LIN {X 0,Y 541.566,Z 805.844,A -85,B 0,C 180,E1 24079.276,E2 24079.276} C_VEL
LIN {X 0,Y 534.284,Z 830.218,A -85,B 0,C 180,E1 24077.061,E2 24077.061} C_VEL
LIN {X 0,Y 530.559,Z 850.368,A -85,B 0,C 180,E1 24075.119,E2 24075.119} C_VEL
LIN {X 0,Y 529.282,Z 869.4,A -85,B 0,C 180,E1 24073.179,E2 24073.179} C_VEL
LIN {X 0,Y 530.561,Z 887.498,A -85,B 0,C 180,E1 24071.24,E2 24071.24} C_VEL
LIN {X 0,Y 533.862,Z 903.063,A -85,B 0,C 180,E1 24069.497,E2 24069.497} C_VEL
LIN {X 0,Y 539.786,Z 919.194,A -85,B 0,C 180,E1 24067.637,E2 24067.637} C_VEL
LIN {X 0,Y 545.938,Z 931.026,A -85,B 0,C 180,E1 24066.25,E2 24066.25} C_VEL
LIN {X 0,Y 535.777,Z 951.59,A -85,B 0,C 180,E1 24065.476,E2 24065.476} C_VEL
LIN {X 0,Y 524.83,Z 974.952,A -85,B 0,C 180,E1 24064.531,E2 24064.531} C_VEL
LIN {X 0,Y 514.891,Z 1001.395,A -85,B 0,C 180,E1 24063.294,E2 24063.294} C_VEL
LIN {X 0,Y 512.272,Z 1027.243,A -85,B 0,C 180,E1 24062.958,E2 24062.958} C_VEL
LIN {X 0,Y 510.91,Z 1051.218,A -85,B 0,C 180,E1 24062.455,E2 24062.455} C_VEL
LIN {X 0,Y 509.239,Z 1078.179,A -85,B 0,C 180,E1 24061.802,E2 24061.802} C_VEL
LIN {X 0,Y 507.496,Z 1100.809,A -85,B 0,C 180,E1 24061.043,E2 24061.043} C_VEL
LIN {X 0,Y 505.536,Z 1122.381,A -85,B 0,C 180,E1 24060.112,E2 24060.112} C_VEL
LIN {X 0,Y 503.367,Z 1143.225,A -85,B 0,C 180,E1 24058.989,E2 24058.989} C_VEL
LIN {X 0,Y 501.157,Z 1162.938,A -85,B 0,C 180,E1 24057.7,E2 24057.7} C_VEL
LIN {X 0,Y 498.803,Z 1182.648,A -85,B 0,C 180,E1 24056.166,E2 24056.166} C_VEL
LIN {X 0,Y 496.617,Z 1200.724,A -85,B 0,C 180,E1 24054.502,E2 24054.502} C_VEL
LIN {X 0,Y 494.521,Z 1217.819,A -85,B 0,C 180,E1 24052.653,E2 24052.653} C_VEL
LIN {X 0,Y 492.705,Z 1233.253,A -85,B 0,C 180,E1 24050.676,E2 24050.676} C_VEL
LIN {X 0,Y 491.203,Z 1246.856,A -85,B 0,C 180,E1 24048.636,E2 24048.636} C_VEL
LIN {X 0,Y 489.996,Z 1259.291,A -85,B 0,C 180,E1 24046.445,E2 24046.445} C_VEL
LIN {X 0,Y 489.117,Z 1269.986,A -85,B 0,C 180,E1 24044.198,E2 24044.198} C_VEL
LIN {X 0,Y 488.558,Z 1278.843,A -85,B 0,C 180,E1 24041.928,E2 24041.928} C_VEL
LIN {X 0,Y 488.232,Z 1286.686,A -85,B 0,C 180,E1 24039.428,E2 24039.428} C_VEL
LIN {X 0,Y 488.136,Z 1292.402,A -85,B 0,C 180,E1 24037.058,E2 24037.058} C_VEL
LIN {X 0,Y 488.13,Z 1296.322,A -85,B 0,C 180,E1 24034.698,E2 24034.698} C_VEL
LIN {X 0,Y 488.17,Z 1298.785,A -85,B 0,C 180,E1 24032.229,E2 24032.229} C_VEL
LIN {X 0,Y 488.204,Z 1299.536,A -85,B 0,C 180,E1 24029.998,E2 24029.998} C_VEL
LIN {X 0,Y 488.169,Z 1298.744,A -85,B 0,C 180,E1 24027.651,E2 24027.651} C_VEL
LIN {X 0,Y 488.128,Z 1296.475,A -85,B 0,C 180,E1 24025.299,E2 24025.299} C_VEL
LIN {X 0,Y 488.129,Z 1292.488,A -85,B 0,C 180,E1 24022.939,E2 24022.939} C_VEL
LIN {X 0,Y 488.239,Z 1286.593,A -85,B 0,C 180,E1 24020.45,E2 24020.45} C_VEL
LIN {X 0,Y 488.572,Z 1279.108,A -85,B 0,C 180,E1 24018.031,E2 24018.031} C_VEL
LIN {X 0,Y 489.169,Z 1269.857,A -85,B 0,C 180,E1 24015.671,E2 24015.671} C_VEL
LIN {X 0,Y 490.098,Z 1259.114,A -85,B 0,C 180,E1 24013.402,E2 24013.402} C_VEL
LIN {X 0,Y 491.35,Z 1247.043,A -85,B 0,C 180,E1 24011.243,E2 24011.243} C_VEL
LIN {X 0,Y 493.006,Z 1232.741,A -85,B 0,C 180,E1 24009.085,E2 24009.085} C_VEL
LIN {X 0,Y 494.933,Z 1217.32,A -85,B 0,C 180,E1 24007.108,E2 24007.108} C_VEL
LIN {X 0,Y 497.21,Z 1200.018,A -85,B 0,C 180,E1 24005.209,E2 24005.209} C_VEL
LIN {X 0,Y 499.657,Z 1181.743,A -85,B 0,C 180,E1 24003.495,E2 24003.495} C_VEL
LIN {X 0,Y 502.296,Z 1161.907,A -85,B 0,C 180,E1 24001.913,E2 24001.913} C_VEL
LIN {X 0,Y 504.977,Z 1141.094,A -85,B 0,C 180,E1 24000.524,E2 24000.524} C_VEL
LIN {X 0,Y 507.637,Z 1119.561,A -85,B 0,C 180,E1 23999.325,E2 23999.325} C_VEL
LIN {X 0,Y 510.395,Z 1095.576,A -85,B 0,C 180,E1 23998.237,E2 23998.237} C_VEL
LIN {X 0,Y 513.002,Z 1071.055,A -85,B 0,C 180,E1 23997.372,E2 23997.372} C_VEL
LIN {X 0,Y 515.293,Z 1044.929,A -85,B 0,C 180,E1 23996.682,E2 23996.682} C_VEL
LIN {X 0,Y 517.326,Z 1019.828,A -85,B 0,C 180,E1 23996.175,E2 23996.175} C_VEL
LIN {X 0,Y 521.032,Z 993.326,A -85,B 0,C 180,E1 23995.793,E2 23995.793} C_VEL
LIN {X 0,Y 524.148,Z 975.151,A -85,B 0,C 180,E1 23995.554,E2 23995.554} C_VEL
LIN {X 0,Y 533.694,Z 955.512,A -85,B 0,C 180,E1 23994.69,E2 23994.69} C_VEL
LIN {X 0,Y 544.849,Z 933.457,A -85,B 0,C 180,E1 23993.776,E2 23993.776} C_VEL
LIN {X 0,Y 546.068,Z 931,A -85,B 0,C 180,E1 23993.676,E2 23993.676} C_VEL
LIN {X 0,Y 537.386,Z 914.874,A -85,B 0,C 180,E1 23992.085,E2 23992.085} C_VEL
LIN {X 0,Y 530.315,Z 896.626,A -85,B 0,C 180,E1 23990.373,E2 23990.373} C_VEL
LIN {X 0,Y 525.51,Z 877.608,A -85,B 0,C 180,E1 23988.681,E2 23988.681} C_VEL
LIN {X 0,Y 522.701,Z 857.001,A -85,B 0,C 180,E1 23986.949,E2 23986.949} C_VEL
LIN {X 0,Y 522.061,Z 833.291,A -85,B 0,C 180,E1 23985.079,E2 23985.079} C_VEL
LIN {X 0,Y 523.719,Z 807.291,A -85,B 0,C 180,E1 23983.17,E2 23983.17} C_VEL
LIN {X 0,Y 524.25,Z 804.145,A -85,B 0,C 180,E1 23982.911,E2 23982.911} C_VEL
LIN {X 0,Y 528.322,Z 794.484,A -85,B 0,C 180,E1 23981.908,E2 23981.908} C_VEL
LIN {X 0,Y 533.971,Z 781.731,A -85,B 0,C 180,E1 23980.903,E2 23980.903} C_VEL
LIN {X 0,Y 539.483,Z 772.496,A -85,B 0,C 180,E1 23979.906,E2 23979.906} C_VEL
LIN {X 0,Y 543.178,Z 766.2,A -85,B 0,C 180,E1 23979.362,E2 23979.362} C_VEL
LIN {X 0,Y 544.157,Z 765.715,A -85,B 0,C 180,E1 23979.153,E2 23979.153} C_VEL
LIN {X 0,Y 533.304,Z 844.029,A -85,B 0,C 180,E1 23977.238,E2 23977.238} C_VEL
LIN {X 0,Y 525.102,Z 918.826,A -85,B 0,C 180,E1 23975.459,E2 23975.459} C_VEL
LIN {X 0,Y 519.129,Z 989.306,A -85,B 0,C 180,E1 23973.885,E2 23973.885} C_VEL
LIN {X 0,Y 516.543,Z 1024.668,A -85,B 0,C 180,E1 23973.074,E2 23973.074} C_VEL
LIN {X 0,Y 514.57,Z 1047.862,A -85,B 0,C 180,E1 23972.334,E2 23972.334} C_VEL
LIN {X 0,Y 512.272,Z 1070.268,A -85,B 0,C 180,E1 23971.41,E2 23971.41} C_VEL
LIN {X 0,Y 509.852,Z 1091.172,A -85,B 0,C 180,E1 23970.338,E2 23970.338} C_VEL
LIN {X 0,Y 507.242,Z 1111.614,A -85,B 0,C 180,E1 23969.072,E2 23969.072} C_VEL
LIN {X 0,Y 504.447,Z 1131.853,A -85,B 0,C 180,E1 23967.57,E2 23967.57} C_VEL
LIN {X 0,Y 501.847,Z 1149.75,A -85,B 0,C 180,E1 23965.998,E2 23965.998} C_VEL
LIN {X 0,Y 499.264,Z 1166.786,A -85,B 0,C 180,E1 23964.24,E2 23964.24} C_VEL
LIN {X 0,Y 496.866,Z 1182.221,A -85,B 0,C 180,E1 23962.355,E2 23962.355} C_VEL
LIN {X 0,Y 494.645,Z 1196.64,A -85,B 0,C 180,E1 23960.289,E2 23960.289} C_VEL
LIN {X 0,Y 492.724,Z 1209.621,A -85,B 0,C 180,E1 23958.089,E2 23958.089} C_VEL
LIN {X 0,Y 491.188,Z 1220.813,A -85,B 0,C 180,E1 23955.83,E2 23955.83} C_VEL
LIN {X 0,Y 489.975,Z 1230.462,A -85,B 0,C 180,E1 23953.453,E2 23953.453} C_VEL
LIN {X 0,Y 489.147,Z 1238.236,A -85,B 0,C 180,E1 23951.078,E2 23951.078} C_VEL
LIN {X 0,Y 488.589,Z 1244.598,A -85,B 0,C 180,E1 23948.592,E2 23948.592} C_VEL
LIN {X 0,Y 488.284,Z 1249.232,A -85,B 0,C 180,E1 23946.113,E2 23946.113} C_VEL
LIN {X 0,Y 488.119,Z 1252.089,A -85,B 0,C 180,E1 23943.641,E2 23943.641} C_VEL
LIN {X 0,Y 488.06,Z 1253.398,A -85,B 0,C 180,E1 23941.057,E2 23941.057} C_VEL
LIN {X 0,Y 488.043,Z 1253.116,A -85,B 0,C 180,E1 23938.709,E2 23938.709} C_VEL
LIN {X 0,Y 488.063,Z 1251.244,A -85,B 0,C 180,E1 23936.359,E2 23936.359} C_VEL
LIN {X 0,Y 488.172,Z 1247.532,A -85,B 0,C 180,E1 23933.768,E2 23933.768} C_VEL
LIN {X 0,Y 488.412,Z 1242.589,A -85,B 0,C 180,E1 23931.405,E2 23931.405} C_VEL
LIN {X 0,Y 488.829,Z 1235.88,A -85,B 0,C 180,E1 23929.034,E2 23929.034} C_VEL
LIN {X 0,Y 489.515,Z 1227.438,A -85,B 0,C 180,E1 23926.655,E2 23926.655} C_VEL
LIN {X 0,Y 490.493,Z 1217.656,A -85,B 0,C 180,E1 23924.39,E2 23924.39} C_VEL
LIN {X 0,Y 491.82,Z 1205.828,A -85,B 0,C 180,E1 23922.122,E2 23922.122} C_VEL
LIN {X 0,Y 493.439,Z 1192.468,A -85,B 0,C 180,E1 23919.973,E2 23919.973} C_VEL
LIN {X 0,Y 495.407,Z 1177.135,A -85,B 0,C 180,E1 23917.884,E2 23917.884} C_VEL
LIN {X 0,Y 497.536,Z 1160.752,A -85,B 0,C 180,E1 23915.986,E2 23915.986} C_VEL
LIN {X 0,Y 499.787,Z 1143.375,A -85,B 0,C 180,E1 23914.269,E2 23914.269} C_VEL
LIN {X 0,Y 502.142,Z 1124.233,A -85,B 0,C 180,E1 23912.678,E2 23912.678} C_VEL
LIN {X 0,Y 504.346,Z 1104.962,A -85,B 0,C 180,E1 23911.329,E2 23911.329} C_VEL
LIN {X 0,Y 506.56,Z 1084.006,A -85,B 0,C 180,E1 23910.105,E2 23910.105} C_VEL
LIN {X 0,Y 508.541,Z 1062.738,A -85,B 0,C 180,E1 23909.091,E2 23909.091} C_VEL
LIN {X 0,Y 510.231,Z 1040.93,A -85,B 0,C 180,E1 23908.268,E2 23908.268} C_VEL
LIN {X 0,Y 511.616,Z 1018.365,A -85,B 0,C 180,E1 23907.63,E2 23907.63} C_VEL
LIN {X 0,Y 512.786,Z 991.425,A -85,B 0,C 180,E1 23907.106,E2 23907.106} C_VEL
LIN {X 0,Y 520.948,Z 782.107,A -85,B 0,C 180,E1 23903.551,E2 23903.551} C_VEL
LIN {X 0,Y 522.188,Z 749.349,A -85,B 0,C 180,E1 23902.975,E2 23902.975} C_VEL
LIN {X 0,Y 520.213,Z 740.745,A -85,B 0,C 180,E1 23902.658,E2 23902.658} C_VEL
LIN {X 0,Y 504.116,Z 709.471,A -85,B 0,C 180,E1 23900.787,E2 23900.787} C_VEL
LIN {X 0,Y 502.649,Z 706.502,A -85,B 0,C 180,E1 23900.593,E2 23900.593} C_VEL
LIN {X 0,Y 494.887,Z 684.827,A -85,B 0,C 180,E1 23897.689,E2 23897.689} C_VEL
LIN {X 0,Y 489.992,Z 671.636,A -85,B 0,C 180,E1 23895.831,E2 23895.831} C_VEL
LIN {X 0,Y 489.982,Z 671.63,A -85,B 0,C 180,E1 23892.203,E2 23892.203} C_VEL
LIN {X 0,Y 489.989,Z 671.636,A -85,B 0,C 180,E1 23888.642,E2 23888.642} C_VEL
LIN {X 0,Y 489.982,Z 671.635,A -85,B 0,C 180,E1 23884.991,E2 23884.991} C_VEL
LIN {X 0,Y 489.985,Z 671.63,A -85,B 0,C 180,E1 23881.461,E2 23881.461} C_VEL
LIN {X 0,Y 489.986,Z 671.63,A -85,B 0,C 180,E1 23877.861,E2 23877.861} C_VEL
LIN {X 0,Y 489.984,Z 671.633,A -85,B 0,C 180,E1 23874.217,E2 23874.217} C_VEL
LIN {X 0,Y 489.996,Z 671.633,A -85,B 0,C 180,E1 23870.504,E2 23870.504} C_VEL
LIN {X 0,Y 489.983,Z 671.633,A -85,B 0,C 180,E1 23866.968,E2 23866.968} C_VEL
LIN {X 0,Y 489.989,Z 671.623,A -85,B 0,C 180,E1 23863.333,E2 23863.333} C_VEL
LIN {X 0,Y 489.982,Z 671.632,A -85,B 0,C 180,E1 23860.024,E2 23860.024} C_VEL
LIN {X 0,Y 489,Z 671.759,A -85,B 0,C 180,E1 23859.123,E2 23859.123} C_VEL
LIN {X 0,Y 482.504,Z 672.571,A -85,B 0,C 180,E1 23856.524,E2 23856.524} C_VEL
LIN {X 0,Y 482.057,Z 672.624,A -85,B 0,C 180,E1 23855.929,E2 23855.929} C_VEL
LIN {X 0,Y 482.048,Z 672.623,A -85,B 0,C 180,E1 23852.26,E2 23852.26} C_VEL
LIN {X 0,Y 482.058,Z 672.617,A -85,B 0,C 180,E1 23848.694,E2 23848.694} C_VEL
LIN {X 0,Y 482.054,Z 672.617,A -85,B 0,C 180,E1 23845.004,E2 23845.004} C_VEL
LIN {X 0,Y 482.046,Z 672.619,A -85,B 0,C 180,E1 23841.413,E2 23841.413} C_VEL
LIN {X 0,Y 482.057,Z 672.621,A -85,B 0,C 180,E1 23837.787,E2 23837.787} C_VEL
LIN {X 0,Y 482.051,Z 672.626,A -85,B 0,C 180,E1 23834.235,E2 23834.235} C_VEL
LIN {X 0,Y 482.05,Z 672.62,A -85,B 0,C 180,E1 23830.619,E2 23830.619} C_VEL
LIN {X 0,Y 482.05,Z 672.62,A -85,B 0,C 180,E1 23826.921,E2 23826.921} C_VEL
LIN {X 0,Y 482.054,Z 672.62,A -85,B 0,C 180,E1 23823.38,E2 23823.38} C_VEL
LIN {X 0,Y 482.055,Z 672.625,A -85,B 0,C 180,E1 23819.735,E2 23819.735} C_VEL
LIN {X 0,Y 482.045,Z 672.625,A -85,B 0,C 180,E1 23816.069,E2 23816.069} C_VEL
LIN {X 0,Y 482.049,Z 672.631,A -85,B 0,C 180,E1 23814.933,E2 23814.933} C_VEL
LIN {X 0,Y 483.508,Z 676.316,A -85,B 0,C 180,E1 23814.363,E2 23814.363} C_VEL
LIN {X 0,Y 491.928,Z 697.055,A -85,B 0,C 180,E1 23811.244,E2 23811.244} C_VEL
LIN {X 0,Y 499.705,Z 717.712,A -85,B 0,C 180,E1 23808.373,E2 23808.373} C_VEL
LIN {X 0,Y 507.183,Z 739.721,A -85,B 0,C 180,E1 23805.534,E2 23805.534} C_VEL
LIN {X 0,Y 508.069,Z 743.311,A -85,B 0,C 180,E1 23805.112,E2 23805.112} C_VEL
LIN {X 0,Y 503.975,Z 782.712,A -85,B 0,C 180,E1 23801.655,E2 23801.655} C_VEL
LIN {X 0,Y 499.66,Z 827.724,A -85,B 0,C 180,E1 23797.76,E2 23797.76} C_VEL
LIN {X 0,Y 495.715,Z 873.661,A -85,B 0,C 180,E1 23793.829,E2 23793.829} C_VEL
LIN {X 0,Y 493.014,Z 910.23,A -85,B 0,C 180,E1 23790.759,E2 23790.759} C_VEL
LIN {X 0,Y 493.892,Z 921.522,A -85,B 0,C 180,E1 23790.465,E2 23790.465} C_VEL
LIN {X 0,Y 489.136,Z 1043.911,A -85,B 0,C 180,E1 23787.805,E2 23787.805} C_VEL
LIN {X 0,Y 488.638,Z 1063.737,A -85,B 0,C 180,E1 23787.27,E2 23787.27} C_VEL
LIN {X 0,Y 487.968,Z 1080.648,A -85,B 0,C 180,E1 23786.576,E2 23786.576} C_VEL
LIN {X 0,Y 487.143,Z 1096.335,A -85,B 0,C 180,E1 23785.706,E2 23785.706} C_VEL
LIN {X 0,Y 486.16,Z 1111.359,A -85,B 0,C 180,E1 23784.629,E2 23784.629} C_VEL
LIN {X 0,Y 485.185,Z 1125.295,A -85,B 0,C 180,E1 23783.373,E2 23783.373} C_VEL
LIN {X 0,Y 484.172,Z 1138.491,A -85,B 0,C 180,E1 23781.891,E2 23781.891} C_VEL
LIN {X 0,Y 483.29,Z 1149.578,A -85,B 0,C 180,E1 23780.339,E2 23780.339} C_VEL
LIN {X 0,Y 482.529,Z 1159.535,A -85,B 0,C 180,E1 23778.61,E2 23778.61} C_VEL
LIN {X 0,Y 481.961,Z 1167.806,A -85,B 0,C 180,E1 23776.761,E2 23776.761} C_VEL
LIN {X 0,Y 481.599,Z 1174.114,A -85,B 0,C 180,E1 23774.919,E2 23774.919} C_VEL
LIN {X 0,Y 481.406,Z 1178.815,A -85,B 0,C 180,E1 23772.963,E2 23772.963} C_VEL
LIN {X 0,Y 481.387,Z 1181.744,A -85,B 0,C 180,E1 23771.017,E2 23771.017} C_VEL
LIN {X 0,Y 481.505,Z 1182.896,A -85,B 0,C 180,E1 23769.08,E2 23769.08} C_VEL
LIN {X 0,Y 481.821,Z 1182.327,A -85,B 0,C 180,E1 23767.033,E2 23767.033} C_VEL
LIN {X 0,Y 482.335,Z 1179.829,A -85,B 0,C 180,E1 23764.995,E2 23764.995} C_VEL
LIN {X 0,Y 483.085,Z 1175.772,A -85,B 0,C 180,E1 23763.085,E2 23763.085} C_VEL
LIN {X 0,Y 484.099,Z 1169.809,A -85,B 0,C 180,E1 23761.184,E2 23761.184} C_VEL
LIN {X 0,Y 485.355,Z 1162.471,A -85,B 0,C 180,E1 23759.41,E2 23759.41} C_VEL
LIN {X 0,Y 486.896,Z 1152.972,A -85,B 0,C 180,E1 23757.646,E2 23757.646} C_VEL
LIN {X 0,Y 488.471,Z 1142.752,A -85,B 0,C 180,E1 23756.127,E2 23756.127} C_VEL
LIN {X 0,Y 490.341,Z 1129.503,A -85,B 0,C 180,E1 23754.559,E2 23754.559} C_VEL
LIN {X 0,Y 492.025,Z 1116.045,A -85,B 0,C 180,E1 23753.29,E2 23753.29} C_VEL
LIN {X 0,Y 493.557,Z 1102.443,A -85,B 0,C 180,E1 23752.257,E2 23752.257} C_VEL
LIN {X 0,Y 494.951,Z 1086.956,A -85,B 0,C 180,E1 23751.344,E2 23751.344} C_VEL
LIN {X 0,Y 496.064,Z 1070.675,A -85,B 0,C 180,E1 23750.618,E2 23750.618} C_VEL
LIN {X 0,Y 498.691,Z 1035.572,A -85,B 0,C 180,E1 23749.45,E2 23749.45} C_VEL
LIN {X 0,Y 506.039,Z 961.807,A -85,B 0,C 180,E1 23747.261,E2 23747.261} C_VEL
LIN {X 0,Y 508.879,Z 930.354,A -85,B 0,C 180,E1 23746.405,E2 23746.405} C_VEL
LIN {X 0,Y 515.809,Z 892.887,A -85,B 0,C 180,E1 23742.747,E2 23742.747} C_VEL
LIN {X 0,Y 524.292,Z 856.411,A -85,B 0,C 180,E1 23739.048,E2 23739.048} C_VEL
LIN {X 0,Y 534.212,Z 822.336,A -85,B 0,C 180,E1 23735.448,E2 23735.448} C_VEL
LIN {X 0,Y 544.197,Z 794.857,A -85,B 0,C 180,E1 23732.418,E2 23732.418} C_VEL
LIN {X 0,Y 545.803,Z 790.745,A -85,B 0,C 180,E1 23731.913,E2 23731.913} C_VEL
LIN {X 0,Y 545.524,Z 785.166,A -85,B 0,C 180,E1 23730.096,E2 23730.096} C_VEL
LIN {X 0,Y 545.538,Z 781.595,A -85,B 0,C 180,E1 23728.386,E2 23728.386} C_VEL
LIN {X 0,Y 545.664,Z 780.156,A -85,B 0,C 180,E1 23727.251,E2 23727.251} C_VEL
LIN {X 0,Y 546.549,Z 778.935,A -85,B 0,C 180,E1 23725.408,E2 23725.408} C_VEL
LIN {X 0,Y 546.702,Z 780.204,A -85,B 0,C 180,E1 23724.178,E2 23724.178} C_VEL
LIN {X 0,Y 547.288,Z 782.485,A -85,B 0,C 180,E1 23722.8,E2 23722.8} C_VEL
LIN {X 0,Y 547.557,Z 784.121,A -85,B 0,C 180,E1 23722.162,E2 23722.162} C_VEL
LIN {X 0,Y 536.082,Z 811.403,A -85,B 0,C 180,E1 23719.668,E2 23719.668} C_VEL
LIN {X 0,Y 528.965,Z 834.107,A -85,B 0,C 180,E1 23717.559,E2 23717.559} C_VEL
LIN {X 0,Y 524.725,Z 855.419,A -85,B 0,C 180,E1 23715.45,E2 23715.45} C_VEL
LIN {X 0,Y 523.335,Z 873.067,A -85,B 0,C 180,E1 23713.604,E2 23713.604} C_VEL
LIN {X 0,Y 524.335,Z 891.469,A -85,B 0,C 180,E1 23711.574,E2 23711.574} C_VEL
LIN {X 0,Y 527.672,Z 907.787,A -85,B 0,C 180,E1 23709.706,E2 23709.706} C_VEL
LIN {X 0,Y 533.253,Z 923.34,A -85,B 0,C 180,E1 23707.869,E2 23707.869} C_VEL
LIN {X 0,Y 538.17,Z 933.25,A -85,B 0,C 180,E1 23706.683,E2 23706.683} C_VEL
LIN {X 0,Y 519.32,Z 972.34,A -85,B 0,C 180,E1 23705.145,E2 23705.145} C_VEL
LIN {X 0,Y 509.067,Z 998.406,A -85,B 0,C 180,E1 23703.903,E2 23703.903} C_VEL
LIN {X 0,Y 508.485,Z 1000.854,A -85,B 0,C 180,E1 23703.828,E2 23703.828} C_VEL
LIN {X 0,Y 505.727,Z 1027.324,A -85,B 0,C 180,E1 23703.476,E2 23703.476} C_VEL
LIN {X 0,Y 504.12,Z 1052.636,A -85,B 0,C 180,E1 23702.917,E2 23702.917} C_VEL
LIN {X 0,Y 501.019,Z 1090.242,A -85,B 0,C 180,E1 23701.787,E2 23701.787} C_VEL
LIN {X 0,Y 499.075,Z 1112.286,A -85,B 0,C 180,E1 23700.921,E2 23700.921} C_VEL
LIN {X 0,Y 496.958,Z 1133.246,A -85,B 0,C 180,E1 23699.889,E2 23699.889} C_VEL
LIN {X 0,Y 494.621,Z 1154.026,A -85,B 0,C 180,E1 23698.624,E2 23698.624} C_VEL
LIN {X 0,Y 492.369,Z 1172.844,A -85,B 0,C 180,E1 23697.252,E2 23697.252} C_VEL
LIN {X 0,Y 490.008,Z 1191.704,A -85,B 0,C 180,E1 23695.63,E2 23695.63} C_VEL
LIN {X 0,Y 487.837,Z 1209.04,A -85,B 0,C 180,E1 23693.877,E2 23693.877} C_VEL
LIN {X 0,Y 485.793,Z 1225.327,A -85,B 0,C 180,E1 23691.934,E2 23691.934} C_VEL
LIN {X 0,Y 484.085,Z 1239.64,A -85,B 0,C 180,E1 23689.924,E2 23689.924} C_VEL
LIN {X 0,Y 482.589,Z 1253.581,A -85,B 0,C 180,E1 23687.619,E2 23687.619} C_VEL
LIN {X 0,Y 481.533,Z 1264.833,A -85,B 0,C 180,E1 23685.412,E2 23685.412} C_VEL
LIN {X 0,Y 480.814,Z 1274.617,A -85,B 0,C 180,E1 23683.099,E2 23683.099} C_VEL
LIN {X 0,Y 480.359,Z 1282.746,A -85,B 0,C 180,E1 23680.736,E2 23680.736} C_VEL
LIN {X 0,Y 480.177,Z 1289.198,A -85,B 0,C 180,E1 23678.38,E2 23678.38} C_VEL
LIN {X 0,Y 480.131,Z 1293.831,A -85,B 0,C 180,E1 23676.095,E2 23676.095} C_VEL
LIN {X 0,Y 480.158,Z 1297.253,A -85,B 0,C 180,E1 23673.58,E2 23673.58} C_VEL
LIN {X 0,Y 480.2,Z 1298.945,A -85,B 0,C 180,E1 23671.191,E2 23671.191} C_VEL
LIN {X 0,Y 480.199,Z 1298.931,A -85,B 0,C 180,E1 23668.805,E2 23668.805} C_VEL
LIN {X 0,Y 480.15,Z 1297.3,A -85,B 0,C 180,E1 23666.297,E2 23666.297} C_VEL
LIN {X 0,Y 480.123,Z 1294.316,A -85,B 0,C 180,E1 23664.022,E2 23664.022} C_VEL
LIN {X 0,Y 480.176,Z 1289.39,A -85,B 0,C 180,E1 23661.539,E2 23661.539} C_VEL
LIN {X 0,Y 480.385,Z 1282.817,A -85,B 0,C 180,E1 23659.08,E2 23659.08} C_VEL
LIN {X 0,Y 480.883,Z 1274.587,A -85,B 0,C 180,E1 23656.683,E2 23656.683} C_VEL
LIN {X 0,Y 481.68,Z 1264.723,A -85,B 0,C 180,E1 23654.343,E2 23654.343} C_VEL
LIN {X 0,Y 482.873,Z 1253.047,A -85,B 0,C 180,E1 23652.028,E2 23652.028} C_VEL
LIN {X 0,Y 484.425,Z 1239.949,A -85,B 0,C 180,E1 23649.835,E2 23649.835} C_VEL
LIN {X 0,Y 486.299,Z 1225.36,A -85,B 0,C 180,E1 23647.769,E2 23647.769} C_VEL
LIN {X 0,Y 488.636,Z 1208.366,A -85,B 0,C 180,E1 23645.712,E2 23645.712} C_VEL
LIN {X 0,Y 491.189,Z 1190.401,A -85,B 0,C 180,E1 23643.861,E2 23643.861} C_VEL
LIN {X 0,Y 493.916,Z 1171.292,A -85,B 0,C 180,E1 23642.183,E2 23642.183} C_VEL
LIN {X 0,Y 496.811,Z 1150.622,A -85,B 0,C 180,E1 23640.653,E2 23640.653} C_VEL
LIN {X 0,Y 499.711,Z 1129.034,A -85,B 0,C 180,E1 23639.319,E2 23639.319} C_VEL
LIN {X 0,Y 502.592,Z 1106.705,A -85,B 0,C 180,E1 23638.182,E2 23638.182} C_VEL
LIN {X 0,Y 505.487,Z 1082.225,A -85,B 0,C 180,E1 23637.179,E2 23637.179} C_VEL
LIN {X 0,Y 508.225,Z 1056.68,A -85,B 0,C 180,E1 23636.386,E2 23636.386} C_VEL
LIN {X 0,Y 510.933,Z 1024.635,A -85,B 0,C 180,E1 23635.65,E2 23635.65} C_VEL
LIN {X 0,Y 514.827,Z 996.352,A -85,B 0,C 180,E1 23635.208,E2 23635.208} C_VEL
LIN {X 0,Y 519.537,Z 969.212,A -85,B 0,C 180,E1 23634.88,E2 23634.88} C_VEL
LIN {X 0,Y 537.73,Z 932.636,A -85,B 0,C 180,E1 23633.336,E2 23633.336} C_VEL
LIN {X 0,Y 529.347,Z 916.206,A -85,B 0,C 180,E1 23631.715,E2 23631.715} C_VEL
LIN {X 0,Y 522.658,Z 898.007,A -85,B 0,C 180,E1 23629.998,E2 23629.998} C_VEL
LIN {X 0,Y 518.027,Z 878.41,A -85,B 0,C 180,E1 23628.246,E2 23628.246} C_VEL
LIN {X 0,Y 515.497,Z 857.573,A -85,B 0,C 180,E1 23626.481,E2 23626.481} C_VEL
LIN {X 0,Y 515.175,Z 835.423,A -85,B 0,C 180,E1 23624.695,E2 23624.695} C_VEL
LIN {X 0,Y 518.021,Z 825.712,A -85,B 0,C 180,E1 23623.627,E2 23623.627} C_VEL
LIN {X 0,Y 522.541,Z 812.796,A -85,B 0,C 180,E1 23622.525,E2 23622.525} C_VEL
LIN {X 0,Y 524.019,Z 809.062,A -85,B 0,C 180,E1 23622.208,E2 23622.208} C_VEL
LIN {X 0,Y 528.795,Z 798.967,A -85,B 0,C 180,E1 23621.185,E2 23621.185} C_VEL
LIN {X 0,Y 535.113,Z 786.094,A -85,B 0,C 180,E1 23620.159,E2 23620.159} C_VEL
LIN {X 0,Y 538.572,Z 781.035,A -85,B 0,C 180,E1 23619.558,E2 23619.558} C_VEL
LIN {X 0,Y 527.139,Z 859.43,A -85,B 0,C 180,E1 23617.603,E2 23617.603} C_VEL
LIN {X 0,Y 518.849,Z 931.026,A -85,B 0,C 180,E1 23615.863,E2 23615.863} C_VEL
LIN {X 0,Y 512.679,Z 999.044,A -85,B 0,C 180,E1 23614.3,E2 23614.3} C_VEL
LIN {X 0,Y 510.303,Z 1028.403,A -85,B 0,C 180,E1 23613.572,E2 23613.572} C_VEL
LIN {X 0,Y 508.125,Z 1051.214,A -85,B 0,C 180,E1 23612.799,E2 23612.799} C_VEL
LIN {X 0,Y 505.708,Z 1072.946,A -85,B 0,C 180,E1 23611.865,E2 23611.865} C_VEL
LIN {X 0,Y 502.906,Z 1095.399,A -85,B 0,C 180,E1 23610.663,E2 23610.663} C_VEL
LIN {X 0,Y 500.07,Z 1115.817,A -85,B 0,C 180,E1 23609.332,E2 23609.332} C_VEL
LIN {X 0,Y 497.156,Z 1135.333,A -85,B 0,C 180,E1 23607.814,E2 23607.814} C_VEL
LIN {X 0,Y 494.34,Z 1153.27,A -85,B 0,C 180,E1 23606.164,E2 23606.164} C_VEL
LIN {X 0,Y 491.659,Z 1169.793,A -85,B 0,C 180,E1 23604.384,E2 23604.384} C_VEL
LIN {X 0,Y 489.193,Z 1184.954,A -85,B 0,C 180,E1 23602.471,E2 23602.471} C_VEL
LIN {X 0,Y 486.825,Z 1199.39,A -85,B 0,C 180,E1 23600.311,E2 23600.311} C_VEL
LIN {X 0,Y 484.888,Z 1211.617,A -85,B 0,C 180,E1 23598.142,E2 23598.142} C_VEL
LIN {X 0,Y 483.217,Z 1223.015,A -85,B 0,C 180,E1 23595.728,E2 23595.728} C_VEL
LIN {X 0,Y 482.018,Z 1232.204,A -85,B 0,C 180,E1 23593.37,E2 23593.37} C_VEL
LIN {X 0,Y 481.152,Z 1239.869,A -85,B 0,C 180,E1 23590.901,E2 23590.901} C_VEL
LIN {X 0,Y 480.609,Z 1245.64,A -85,B 0,C 180,E1 23588.494,E2 23588.494} C_VEL
LIN {X 0,Y 480.306,Z 1249.898,A -85,B 0,C 180,E1 23586.095,E2 23586.095} C_VEL
LIN {X 0,Y 480.138,Z 1252.559,A -85,B 0,C 180,E1 23583.701,E2 23583.701} C_VEL
LIN {X 0,Y 480.07,Z 1253.797,A -85,B 0,C 180,E1 23581.193,E2 23581.193} C_VEL
LIN {X 0,Y 480.054,Z 1253.534,A -85,B 0,C 180,E1 23578.807,E2 23578.807} C_VEL
LIN {X 0,Y 480.071,Z 1251.68,A -85,B 0,C 180,E1 23576.418,E2 23576.418} C_VEL
LIN {X 0,Y 480.175,Z 1248.202,A -85,B 0,C 180,E1 23573.904,E2 23573.904} C_VEL
LIN {X 0,Y 480.409,Z 1243.312,A -85,B 0,C 180,E1 23571.502,E2 23571.502} C_VEL
LIN {X 0,Y 480.831,Z 1236.698,A -85,B 0,C 180,E1 23569.092,E2 23569.092} C_VEL
LIN {X 0,Y 481.57,Z 1227.883,A -85,B 0,C 180,E1 23566.553,E2 23566.553} C_VEL
LIN {X 0,Y 482.582,Z 1218.086,A -85,B 0,C 180,E1 23564.251,E2 23564.251} C_VEL
LIN {X 0,Y 483.957,Z 1206.235,A -85,B 0,C 180,E1 23561.946,E2 23561.946} C_VEL
LIN {X 0,Y 485.633,Z 1192.859,A -85,B 0,C 180,E1 23559.763,E2 23559.763} C_VEL
LIN {X 0,Y 487.603,Z 1178.019,A -85,B 0,C 180,E1 23557.705,E2 23557.705} C_VEL
LIN {X 0,Y 489.722,Z 1162.23,A -85,B 0,C 180,E1 23555.835,E2 23555.835} C_VEL
LIN {X 0,Y 492.11,Z 1144.322,A -85,B 0,C 180,E1 23554.032,E2 23554.032} C_VEL
LIN {X 0,Y 494.528,Z 1125.241,A -85,B 0,C 180,E1 23552.418,E2 23552.418} C_VEL
LIN {X 0,Y 496.797,Z 1106.085,A -85,B 0,C 180,E1 23551.05,E2 23551.05} C_VEL
LIN {X 0,Y 499.067,Z 1085.299,A -85,B 0,C 180,E1 23549.809,E2 23549.809} C_VEL
LIN {X 0,Y 501.105,Z 1064.318,A -85,B 0,C 180,E1 23548.782,E2 23548.782} C_VEL
LIN {X 0,Y 502.936,Z 1041.456,A -85,B 0,C 180,E1 23547.901,E2 23547.901} C_VEL
LIN {X 0,Y 504.366,Z 1018.959,A -85,B 0,C 180,E1 23547.253,E2 23547.253} C_VEL
LIN {X 0,Y 505.572,Z 992.417,A -85,B 0,C 180,E1 23546.724,E2 23546.724} C_VEL
LIN {X 0,Y 514.074,Z 784.251,A -85,B 0,C 180,E1 23543.116,E2 23543.116} C_VEL
LIN {X 0,Y 515.433,Z 750.903,A -85,B 0,C 180,E1 23542.519,E2 23542.519} C_VEL
LIN {X 0,Y 513.827,Z 744.191,A -85,B 0,C 180,E1 23542.261,E2 23542.261} C_VEL
LIN {X 0,Y 496.759,Z 710.979,A -85,B 0,C 180,E1 23540.234,E2 23540.234} C_VEL
LIN {X 0,Y 494.51,Z 706.689,A -85,B 0,C 180,E1 23539.937,E2 23539.937} C_VEL
LIN {X 0,Y 486.912,Z 685.592,A -85,B 0,C 180,E1 23537.063,E2 23537.063} C_VEL
LIN {X 0,Y 482.055,Z 672.619,A -85,B 0,C 180,E1 23535.215,E2 23535.215} C_VEL
LIN {X 0,Y 482.056,Z 672.623,A -85,B 0,C 180,E1 23531.588,E2 23531.588} C_VEL
LIN {X 0,Y 482.051,Z 672.622,A -85,B 0,C 180,E1 23527.981,E2 23527.981} C_VEL
LIN {X 0,Y 482.049,Z 672.616,A -85,B 0,C 180,E1 23524.348,E2 23524.348} C_VEL
LIN {X 0,Y 482.056,Z 672.612,A -85,B 0,C 180,E1 23520.821,E2 23520.821} C_VEL
LIN {X 0,Y 482.054,Z 672.625,A -85,B 0,C 180,E1 23517.146,E2 23517.146} C_VEL
LIN {X 0,Y 482.058,Z 672.622,A -85,B 0,C 180,E1 23513.536,E2 23513.536} C_VEL
LIN {X 0,Y 482.057,Z 672.62,A -85,B 0,C 180,E1 23509.889,E2 23509.889} C_VEL
LIN {X 0,Y 482.043,Z 672.624,A -85,B 0,C 180,E1 23506.263,E2 23506.263} C_VEL
LIN {X 0,Y 482.058,Z 672.61,A -85,B 0,C 180,E1 23502.703,E2 23502.703} C_VEL
LIN {X 0,Y 482.041,Z 672.612,A -85,B 0,C 180,E1 23499.072,E2 23499.072} C_VEL
LIN {X 0,Y 482.057,Z 672.624,A -85,B 0,C 180,E1 23495.929,E2 23495.929} C_VEL
LIN {X 0,Y 481.057,Z 672.745,A -85,B 0,C 180,E1 23495.013,E2 23495.013} C_VEL
LIN {X 0,Y 474.551,Z 673.559,A -85,B 0,C 180,E1 23492.372,E2 23492.372} C_VEL
LIN {X 0,Y 474.105,Z 673.611,A -85,B 0,C 180,E1 23491.767,E2 23491.767} C_VEL
LIN {X 0,Y 474.115,Z 673.611,A -85,B 0,C 180,E1 23488.189,E2 23488.189} C_VEL
LIN {X 0,Y 474.103,Z 673.611,A -85,B 0,C 180,E1 23484.434,E2 23484.434} C_VEL
LIN {X 0,Y 474.105,Z 673.611,A -85,B 0,C 180,E1 23480.901,E2 23480.901} C_VEL
LIN {X 0,Y 474.105,Z 673.612,A -85,B 0,C 180,E1 23477.208,E2 23477.208} C_VEL
LIN {X 0,Y 474.105,Z 673.611,A -85,B 0,C 180,E1 23473.659,E2 23473.659} C_VEL
LIN {X 0,Y 474.109,Z 673.605,A -85,B 0,C 180,E1 23470.024,E2 23470.024} C_VEL
LIN {X 0,Y 474.106,Z 673.612,A -85,B 0,C 180,E1 23466.38,E2 23466.38} C_VEL
LIN {X 0,Y 474.112,Z 673.606,A -85,B 0,C 180,E1 23462.767,E2 23462.767} C_VEL
LIN {X 0,Y 474.108,Z 673.612,A -85,B 0,C 180,E1 23459.133,E2 23459.133} C_VEL
LIN {X 0,Y 474.136,Z 673.807,A -85,B 0,C 180,E1 23455.684,E2 23455.684} C_VEL
LIN {X 0,Y 483.221,Z 695.928,A -85,B 0,C 180,E1 23452.233,E2 23452.233} C_VEL
LIN {X 0,Y 490.96,Z 716.135,A -85,B 0,C 180,E1 23449.332,E2 23449.332} C_VEL
LIN {X 0,Y 498.479,Z 737.808,A -85,B 0,C 180,E1 23446.45,E2 23446.45} C_VEL
LIN {X 0,Y 501.006,Z 745.865,A -85,B 0,C 180,E1 23445.438,E2 23445.438} C_VEL
LIN {X 0,Y 496.638,Z 786.335,A -85,B 0,C 180,E1 23441.851,E2 23441.851} C_VEL
LIN {X 0,Y 492.162,Z 831.237,A -85,B 0,C 180,E1 23437.921,E2 23437.921} C_VEL
LIN {X 0,Y 488.15,Z 876.554,A -85,B 0,C 180,E1 23434,E2 23434} C_VEL
LIN {X 0,Y 485.542,Z 910.886,A -85,B 0,C 180,E1 23431.095,E2 23431.095} C_VEL
LIN {X 0,Y 486.413,Z 922.266,A -85,B 0,C 180,E1 23430.792,E2 23430.792} C_VEL
LIN {X 0,Y 481.377,Z 1047.188,A -85,B 0,C 180,E1 23427.995,E2 23427.995} C_VEL
LIN {X 0,Y 480.879,Z 1065.603,A -85,B 0,C 180,E1 23427.466,E2 23427.466} C_VEL
LIN {X 0,Y 480.158,Z 1082.786,A -85,B 0,C 180,E1 23426.731,E2 23426.731} C_VEL
LIN {X 0,Y 479.306,Z 1098.079,A -85,B 0,C 180,E1 23425.849,E2 23425.849} C_VEL
LIN {X 0,Y 478.274,Z 1113.391,A -85,B 0,C 180,E1 23424.716,E2 23424.716} C_VEL
LIN {X 0,Y 477.26,Z 1127.215,A -85,B 0,C 180,E1 23423.423,E2 23423.423} C_VEL
LIN {X 0,Y 476.25,Z 1140.011,A -85,B 0,C 180,E1 23421.945,E2 23421.945} C_VEL
LIN {X 0,Y 475.32,Z 1151.333,A -85,B 0,C 180,E1 23420.31,E2 23420.31} C_VEL
LIN {X 0,Y 474.556,Z 1161.114,A -85,B 0,C 180,E1 23418.552,E2 23418.552} C_VEL
LIN {X 0,Y 473.988,Z 1169.248,A -85,B 0,C 180,E1 23416.672,E2 23416.672} C_VEL
LIN {X 0,Y 473.626,Z 1175.436,A -85,B 0,C 180,E1 23414.792,E2 23414.792} C_VEL
LIN {X 0,Y 473.446,Z 1180.302,A -85,B 0,C 180,E1 23412.664,E2 23412.664} C_VEL
LIN {X 0,Y 473.445,Z 1182.96,A -85,B 0,C 180,E1 23410.711,E2 23410.711} C_VEL
LIN {X 0,Y 473.63,Z 1183.96,A -85,B 0,C 180,E1 23408.621,E2 23408.621} C_VEL
LIN {X 0,Y 473.969,Z 1183.164,A -85,B 0,C 180,E1 23406.663,E2 23406.663} C_VEL
LIN {X 0,Y 474.571,Z 1180.506,A -85,B 0,C 180,E1 23404.592,E2 23404.592} C_VEL
LIN {X 0,Y 475.423,Z 1176.144,A -85,B 0,C 180,E1 23402.619,E2 23402.619} C_VEL
LIN {X 0,Y 476.62,Z 1169.725,A -85,B 0,C 180,E1 23400.601,E2 23400.601} C_VEL
LIN {X 0,Y 478.11,Z 1161.395,A -85,B 0,C 180,E1 23398.682,E2 23398.682} C_VEL
LIN {X 0,Y 479.708,Z 1152.125,A -85,B 0,C 180,E1 23397.013,E2 23397.013} C_VEL
LIN {X 0,Y 481.578,Z 1140.603,A -85,B 0,C 180,E1 23395.355,E2 23395.355} C_VEL
LIN {X 0,Y 483.383,Z 1128.308,A -85,B 0,C 180,E1 23393.944,E2 23393.944} C_VEL
LIN {X 0,Y 485.125,Z 1115.141,A -85,B 0,C 180,E1 23392.718,E2 23392.718} C_VEL
LIN {X 0,Y 486.835,Z 1100.103,A -85,B 0,C 180,E1 23391.615,E2 23391.615} C_VEL
LIN {X 0,Y 488.247,Z 1085.107,A -85,B 0,C 180,E1 23390.749,E2 23390.749} C_VEL
LIN {X 0,Y 489.439,Z 1068.059,A -85,B 0,C 180,E1 23390.015,E2 23390.015} C_VEL
LIN {X 0,Y 492.679,Z 1030.711,A -85,B 0,C 180,E1 23388.754,E2 23388.754} C_VEL
LIN {X 0,Y 499.562,Z 965.705,A -85,B 0,C 180,E1 23386.773,E2 23386.773} C_VEL
LIN {X 0,Y 502.806,Z 932.185,A -85,B 0,C 180,E1 23385.842,E2 23385.842} C_VEL
LIN {X 0,Y 502.958,Z 930.038,A -85,B 0,C 180,E1 23385.67,E2 23385.67} C_VEL
LIN {X 0,Y 511.171,Z 889.858,A -85,B 0,C 180,E1 23381.643,E2 23381.643} C_VEL
LIN {X 0,Y 520.345,Z 854.077,A -85,B 0,C 180,E1 23377.934,E2 23377.934} C_VEL
LIN {X 0,Y 531.007,Z 820.785,A -85,B 0,C 180,E1 23374.336,E2 23374.336} C_VEL
LIN {X 0,Y 540.786,Z 796.114,A -85,B 0,C 180,E1 23371.538,E2 23371.538} C_VEL
LIN {X 0,Y 540.789,Z 790.768,A -85,B 0,C 180,E1 23369.684,E2 23369.684} C_VEL
LIN {X 0,Y 541.037,Z 787.258,A -85,B 0,C 180,E1 23367.821,E2 23367.821} C_VEL
LIN {X 0,Y 541.971,Z 785.498,A -85,B 0,C 180,E1 23365.501,E2 23365.501} C_VEL
LIN {X 0,Y 542.099,Z 786.426,A -85,B 0,C 180,E1 23364.478,E2 23364.478} C_VEL
LIN {X 0,Y 542.625,Z 788.876,A -85,B 0,C 180,E1 23362.925,E2 23362.925} C_VEL
LIN {X 0,Y 542.735,Z 789.681,A -85,B 0,C 180,E1 23362.609,E2 23362.609} C_VEL
LIN {X 0,Y 530.715,Z 817.105,A -85,B 0,C 180,E1 23360.064,E2 23360.064} C_VEL
LIN {X 0,Y 523.324,Z 839.611,A -85,B 0,C 180,E1 23357.915,E2 23357.915} C_VEL
LIN {X 0,Y 519.032,Z 859.867,A -85,B 0,C 180,E1 23355.854,E2 23355.854} C_VEL
LIN {X 0,Y 517.419,Z 878.233,A -85,B 0,C 180,E1 23353.879,E2 23353.879} C_VEL
LIN {X 0,Y 518.202,Z 895.443,A -85,B 0,C 180,E1 23351.932,E2 23351.932} C_VEL
LIN {X 0,Y 521.352,Z 912.027,A -85,B 0,C 180,E1 23349.975,E2 23349.975} C_VEL
LIN {X 0,Y 527.163,Z 928.453,A -85,B 0,C 180,E1 23347.992,E2 23347.992} C_VEL
LIN {X 0,Y 530.472,Z 935.528,A -85,B 0,C 180,E1 23347.125,E2 23347.125} C_VEL
LIN {X 0,Y 512.762,Z 972.302,A -85,B 0,C 180,E1 23345.663,E2 23345.663} C_VEL
LIN {X 0,Y 502.349,Z 999.002,A -85,B 0,C 180,E1 23344.402,E2 23344.402} C_VEL
LIN {X 0,Y 499.28,Z 1027.08,A -85,B 0,C 180,E1 23344.018,E2 23344.018} C_VEL
LIN {X 0,Y 497.514,Z 1052.973,A -85,B 0,C 180,E1 23343.433,E2 23343.433} C_VEL
LIN {X 0,Y 495.266,Z 1075.906,A -85,B 0,C 180,E1 23342.719,E2 23342.719} C_VEL
LIN {X 0,Y 491.861,Z 1110.571,A -85,B 0,C 180,E1 23341.358,E2 23341.358} C_VEL
LIN {X 0,Y 489.612,Z 1132.129,A -85,B 0,C 180,E1 23340.291,E2 23340.291} C_VEL
LIN {X 0,Y 487.205,Z 1152.964,A -85,B 0,C 180,E1 23339.014,E2 23339.014} C_VEL
LIN {X 0,Y 484.799,Z 1172.432,A -85,B 0,C 180,E1 23337.58,E2 23337.58} C_VEL
LIN {X 0,Y 482.363,Z 1191.309,A -85,B 0,C 180,E1 23335.935,E2 23335.935} C_VEL
LIN {X 0,Y 480.174,Z 1208.213,A -85,B 0,C 180,E1 23334.206,E2 23334.206} C_VEL
LIN {X 0,Y 478.054,Z 1224.48,A -85,B 0,C 180,E1 23332.243,E2 23332.243} C_VEL
LIN {X 0,Y 476.291,Z 1238.817,A -85,B 0,C 180,E1 23330.215,E2 23330.215} C_VEL
LIN {X 0,Y 474.736,Z 1252.677,A -85,B 0,C 180,E1 23327.907,E2 23327.907} C_VEL
LIN {X 0,Y 473.632,Z 1263.999,A -85,B 0,C 180,E1 23325.676,E2 23325.676} C_VEL
LIN {X 0,Y 472.864,Z 1273.855,A -85,B 0,C 180,E1 23323.324,E2 23323.324} C_VEL
LIN {X 0,Y 472.374,Z 1282.279,A -85,B 0,C 180,E1 23320.857,E2 23320.857} C_VEL
LIN {X 0,Y 472.182,Z 1288.899,A -85,B 0,C 180,E1 23318.4,E2 23318.4} C_VEL
LIN {X 0,Y 472.137,Z 1293.521,A -85,B 0,C 180,E1 23316.077,E2 23316.077} C_VEL
LIN {X 0,Y 472.17,Z 1296.907,A -85,B 0,C 180,E1 23313.519,E2 23313.519} C_VEL
LIN {X 0,Y 472.211,Z 1298.564,A -85,B 0,C 180,E1 23311.09,E2 23311.09} C_VEL
LIN {X 0,Y 472.207,Z 1298.503,A -85,B 0,C 180,E1 23308.664,E2 23308.664} C_VEL
LIN {X 0,Y 472.152,Z 1296.813,A -85,B 0,C 180,E1 23306.113,E2 23306.113} C_VEL
LIN {X 0,Y 472.128,Z 1293.787,A -85,B 0,C 180,E1 23303.798,E2 23303.798} C_VEL
LIN {X 0,Y 472.183,Z 1288.959,A -85,B 0,C 180,E1 23301.351,E2 23301.351} C_VEL
LIN {X 0,Y 472.415,Z 1282.517,A -85,B 0,C 180,E1 23298.894,E2 23298.894} C_VEL
LIN {X 0,Y 472.956,Z 1274.187,A -85,B 0,C 180,E1 23296.426,E2 23296.426} C_VEL
LIN {X 0,Y 473.87,Z 1263.893,A -85,B 0,C 180,E1 23293.952,E2 23293.952} C_VEL
LIN {X 0,Y 475.245,Z 1251.447,A -85,B 0,C 180,E1 23291.475,E2 23291.475} C_VEL
LIN {X 0,Y 476.981,Z 1237.977,A -85,B 0,C 180,E1 23289.22,E2 23289.22} C_VEL
LIN {X 0,Y 479.146,Z 1222.501,A -85,B 0,C 180,E1 23287.03,E2 23287.03} C_VEL
LIN {X 0,Y 481.63,Z 1205.649,A -85,B 0,C 180,E1 23285.008,E2 23285.008} C_VEL
LIN {X 0,Y 484.311,Z 1187.865,A -85,B 0,C 180,E1 23283.184,E2 23283.184} C_VEL
LIN {X 0,Y 487.352,Z 1167.873,A -85,B 0,C 180,E1 23281.441,E2 23281.441} C_VEL
LIN {X 0,Y 490.364,Z 1147.828,A -85,B 0,C 180,E1 23279.959,E2 23279.959} C_VEL
LIN {X 0,Y 493.653,Z 1125.122,A -85,B 0,C 180,E1 23278.562,E2 23278.562} C_VEL
LIN {X 0,Y 496.896,Z 1101.217,A -85,B 0,C 180,E1 23277.364,E2 23277.364} C_VEL
LIN {X 0,Y 499.903,Z 1077.484,A -85,B 0,C 180,E1 23276.423,E2 23276.423} C_VEL
LIN {X 0,Y 502.697,Z 1052.666,A -85,B 0,C 180,E1 23275.665,E2 23275.665} C_VEL
LIN {X 0,Y 505.53,Z 1022.5,A -85,B 0,C 180,E1 23274.972,E2 23274.972} C_VEL
LIN {X 0,Y 509.647,Z 994.526,A -85,B 0,C 180,E1 23274.532,E2 23274.532} C_VEL
LIN {X 0,Y 514.331,Z 968.49,A -85,B 0,C 180,E1 23274.211,E2 23274.211} C_VEL
LIN {X 0,Y 516.167,Z 960.536,A -85,B 0,C 180,E1 23274.126,E2 23274.126} C_VEL
LIN {X 0,Y 529.544,Z 934.387,A -85,B 0,C 180,E1 23273.008,E2 23273.008} C_VEL
LIN {X 0,Y 521.286,Z 917.348,A -85,B 0,C 180,E1 23271.323,E2 23271.323} C_VEL
LIN {X 0,Y 514.83,Z 898.663,A -85,B 0,C 180,E1 23269.556,E2 23269.556} C_VEL
LIN {X 0,Y 510.508,Z 878.73,A -85,B 0,C 180,E1 23267.762,E2 23267.762} C_VEL
LIN {X 0,Y 508.88,Z 864.729,A -85,B 0,C 180,E1 23266.528,E2 23266.528} C_VEL
LIN {X 0,Y 510.458,Z 854.225,A -85,B 0,C 180,E1 23265.313,E2 23265.313} C_VEL
LIN {X 0,Y 513.701,Z 841.345,A -85,B 0,C 180,E1 23264.11,E2 23264.11} C_VEL
LIN {X 0,Y 517.292,Z 830.883,A -85,B 0,C 180,E1 23262.957,E2 23262.957} C_VEL
LIN {X 0,Y 522.445,Z 817.854,A -85,B 0,C 180,E1 23261.842,E2 23261.842} C_VEL
LIN {X 0,Y 524.123,Z 814.064,A -85,B 0,C 180,E1 23261.513,E2 23261.513} C_VEL
LIN {X 0,Y 529.657,Z 803.429,A -85,B 0,C 180,E1 23260.465,E2 23260.465} C_VEL
LIN {X 0,Y 532.923,Z 797.351,A -85,B 0,C 180,E1 23259.952,E2 23259.952} C_VEL
LIN {X 0,Y 521.452,Z 871.9,A -85,B 0,C 180,E1 23258.055,E2 23258.055} C_VEL
LIN {X 0,Y 512.7,Z 942.896,A -85,B 0,C 180,E1 23256.288,E2 23256.288} C_VEL
LIN {X 0,Y 504.801,Z 1025.887,A -85,B 0,C 180,E1 23254.287,E2 23254.287} C_VEL
LIN {X 0,Y 502.438,Z 1049.203,A -85,B 0,C 180,E1 23253.503,E2 23253.503} C_VEL
LIN {X 0,Y 499.67,Z 1072.397,A -85,B 0,C 180,E1 23252.5,E2 23252.5} C_VEL
LIN {X 0,Y 496.674,Z 1094.757,A -85,B 0,C 180,E1 23251.292,E2 23251.292} C_VEL
LIN {X 0,Y 493.778,Z 1114.338,A -85,B 0,C 180,E1 23250.011,E2 23250.011} C_VEL
LIN {X 0,Y 490.665,Z 1134.045,A -85,B 0,C 180,E1 23248.48,E2 23248.48} C_VEL
LIN {X 0,Y 487.659,Z 1152.189,A -85,B 0,C 180,E1 23246.813,E2 23246.813} C_VEL
LIN {X 0,Y 484.792,Z 1168.909,A -85,B 0,C 180,E1 23245.013,E2 23245.013} C_VEL
LIN {X 0,Y 481.972,Z 1185.05,A -85,B 0,C 180,E1 23242.956,E2 23242.956} C_VEL
LIN {X 0,Y 479.56,Z 1198.757,A -85,B 0,C 180,E1 23240.888,E2 23240.888} C_VEL
LIN {X 0,Y 477.463,Z 1211.161,A -85,B 0,C 180,E1 23238.688,E2 23238.688} C_VEL
LIN {X 0,Y 475.721,Z 1222.216,A -85,B 0,C 180,E1 23236.359,E2 23236.359} C_VEL
LIN {X 0,Y 474.338,Z 1231.793,A -85,B 0,C 180,E1 23233.905,E2 23233.905} C_VEL
LIN {X 0,Y 473.366,Z 1239.474,A -85,B 0,C 180,E1 23231.444,E2 23231.444} C_VEL
LIN {X 0,Y 472.692,Z 1245.96,A -85,B 0,C 180,E1 23228.76,E2 23228.76} C_VEL
LIN {X 0,Y 472.34,Z 1250.411,A -85,B 0,C 180,E1 23226.198,E2 23226.198} C_VEL
LIN {X 0,Y 472.158,Z 1253.038,A -85,B 0,C 180,E1 23223.764,E2 23223.764} C_VEL
LIN {X 0,Y 472.082,Z 1254.216,A -85,B 0,C 180,E1 23221.214,E2 23221.214} C_VEL
LIN {X 0,Y 472.062,Z 1253.895,A -85,B 0,C 180,E1 23218.773,E2 23218.773} C_VEL
LIN {X 0,Y 472.08,Z 1251.989,A -85,B 0,C 180,E1 23216.357,E2 23216.357} C_VEL
LIN {X 0,Y 472.19,Z 1248.426,A -85,B 0,C 180,E1 23213.8,E2 23213.8} C_VEL
LIN {X 0,Y 472.441,Z 1243.481,A -85,B 0,C 180,E1 23211.358,E2 23211.358} C_VEL
LIN {X 0,Y 472.903,Z 1236.554,A -85,B 0,C 180,E1 23208.836,E2 23208.836} C_VEL
LIN {X 0,Y 473.672,Z 1227.828,A -85,B 0,C 180,E1 23206.324,E2 23206.324} C_VEL
LIN {X 0,Y 474.737,Z 1217.899,A -85,B 0,C 180,E1 23203.984,E2 23203.984} C_VEL
LIN {X 0,Y 476.183,Z 1205.95,A -85,B 0,C 180,E1 23201.641,E2 23201.641} C_VEL
LIN {X 0,Y 477.938,Z 1192.403,A -85,B 0,C 180,E1 23199.423,E2 23199.423} C_VEL
LIN {X 0,Y 479.994,Z 1177.365,A -85,B 0,C 180,E1 23197.333,E2 23197.333} C_VEL
LIN {X 0,Y 482.292,Z 1160.79,A -85,B 0,C 180,E1 23195.373,E2 23195.373} C_VEL
LIN {X 0,Y 484.609,Z 1143.911,A -85,B 0,C 180,E1 23193.666,E2 23193.666} C_VEL
LIN {X 0,Y 487.123,Z 1124.708,A -85,B 0,C 180,E1 23192.029,E2 23192.029} C_VEL
LIN {X 0,Y 489.464,Z 1105.37,A -85,B 0,C 180,E1 23190.641,E2 23190.641} C_VEL
LIN {X 0,Y 491.818,Z 1084.34,A -85,B 0,C 180,E1 23189.384,E2 23189.384} C_VEL
LIN {X 0,Y 493.859,Z 1063.726,A -85,B 0,C 180,E1 23188.373,E2 23188.373} C_VEL
LIN {X 0,Y 495.679,Z 1041.688,A -85,B 0,C 180,E1 23187.514,E2 23187.514} C_VEL
LIN {X 0,Y 497.161,Z 1019.155,A -85,B 0,C 180,E1 23186.856,E2 23186.856} C_VEL
LIN {X 0,Y 498.433,Z 992.182,A -85,B 0,C 180,E1 23186.309,E2 23186.309} C_VEL
LIN {X 0,Y 507.566,Z 778.644,A -85,B 0,C 180,E1 23182.537,E2 23182.537} C_VEL
LIN {X 0,Y 508.622,Z 752.27,A -85,B 0,C 180,E1 23182.053,E2 23182.053} C_VEL
LIN {X 0,Y 507.483,Z 747.809,A -85,B 0,C 180,E1 23181.874,E2 23181.874} C_VEL
LIN {X 0,Y 490.92,Z 715.487,A -85,B 0,C 180,E1 23179.868,E2 23179.868} C_VEL
LIN {X 0,Y 486.562,Z 707.242,A -85,B 0,C 180,E1 23179.316,E2 23179.316} C_VEL
LIN {X 0,Y 478.939,Z 686.414,A -85,B 0,C 180,E1 23176.423,E2 23176.423} C_VEL
LIN {X 0,Y 474.11,Z 673.607,A -85,B 0,C 180,E1 23174.573,E2 23174.573} C_VEL
LIN {X 0,Y 474.105,Z 673.616,A -85,B 0,C 180,E1 23170.972,E2 23170.972} C_VEL
LIN {X 0,Y 474.112,Z 673.604,A -85,B 0,C 180,E1 23167.336,E2 23167.336} C_VEL
LIN {X 0,Y 474.106,Z 673.605,A -85,B 0,C 180,E1 23163.689,E2 23163.689} C_VEL
LIN {X 0,Y 474.111,Z 673.607,A -85,B 0,C 180,E1 23159.99,E2 23159.99} C_VEL
LIN {X 0,Y 474.106,Z 673.609,A -85,B 0,C 180,E1 23156.425,E2 23156.425} C_VEL
LIN {X 0,Y 474.112,Z 673.61,A -85,B 0,C 180,E1 23152.704,E2 23152.704} C_VEL
LIN {X 0,Y 474.106,Z 673.607,A -85,B 0,C 180,E1 23149.082,E2 23149.082} C_VEL
LIN {X 0,Y 474.109,Z 673.61,A -85,B 0,C 180,E1 23145.412,E2 23145.412} C_VEL
LIN {X 0,Y 474.105,Z 673.605,A -85,B 0,C 180,E1 23141.806,E2 23141.806} C_VEL
LIN {X 0,Y 474.116,Z 673.596,A -85,B 0,C 180,E1 23138.125,E2 23138.125} C_VEL
LIN {X 0,Y 474.101,Z 673.606,A -85,B 0,C 180,E1 23134.598,E2 23134.598} C_VEL
LIN {X 0,Y 474.105,Z 673.611,A -85,B 0,C 180,E1 23131.767,E2 23131.767} C_VEL
LIN {X 0,Y 473.107,Z 673.734,A -85,B 0,C 180,E1 23130.836,E2 23130.836} C_VEL
LIN {X 0,Y 466.609,Z 674.546,A -85,B 0,C 180,E1 23128.149,E2 23128.149} C_VEL
LIN {X 0,Y 466.167,Z 674.6,A -85,B 0,C 180,E1 23127.534,E2 23127.534} C_VEL
LIN {X 0,Y 466.175,Z 674.6,A -85,B 0,C 180,E1 23123.845,E2 23123.845} C_VEL
LIN {X 0,Y 466.167,Z 674.602,A -85,B 0,C 180,E1 23120.121,E2 23120.121} C_VEL
LIN {X 0,Y 466.177,Z 674.598,A -85,B 0,C 180,E1 23116.482,E2 23116.482} C_VEL
LIN {X 0,Y 466.179,Z 674.595,A -85,B 0,C 180,E1 23112.785,E2 23112.785} C_VEL
LIN {X 0,Y 466.174,Z 674.598,A -85,B 0,C 180,E1 23109.144,E2 23109.144} C_VEL
LIN {X 0,Y 466.177,Z 674.598,A -85,B 0,C 180,E1 23105.548,E2 23105.548} C_VEL
LIN {X 0,Y 466.182,Z 674.599,A -85,B 0,C 180,E1 23101.828,E2 23101.828} C_VEL
LIN {X 0,Y 466.169,Z 674.582,A -85,B 0,C 180,E1 23098.145,E2 23098.145} C_VEL
LIN {X 0,Y 466.169,Z 674.593,A -85,B 0,C 180,E1 23096.514,E2 23096.514} C_VEL
LIN {X 0,Y 467.566,Z 678.219,A -85,B 0,C 180,E1 23095.927,E2 23095.927} C_VEL
LIN {X 0,Y 475.492,Z 697.344,A -85,B 0,C 180,E1 23092.88,E2 23092.88} C_VEL
LIN {X 0,Y 483.225,Z 717.246,A -85,B 0,C 180,E1 23089.948,E2 23089.948} C_VEL
LIN {X 0,Y 490.795,Z 738.959,A -85,B 0,C 180,E1 23087.003,E2 23087.003} C_VEL
LIN {X 0,Y 493.934,Z 748.708,A -85,B 0,C 180,E1 23085.749,E2 23085.749} C_VEL
LIN {X 0,Y 489.34,Z 789.613,A -85,B 0,C 180,E1 23082.084,E2 23082.084} C_VEL
LIN {X 0,Y 484.751,Z 833.914,A -85,B 0,C 180,E1 23078.162,E2 23078.162} C_VEL
LIN {X 0,Y 480.658,Z 878.731,A -85,B 0,C 180,E1 23074.244,E2 23074.244} C_VEL
LIN {X 0,Y 478.074,Z 911.586,A -85,B 0,C 180,E1 23071.434,E2 23071.434} C_VEL
LIN {X 0,Y 478.919,Z 923.147,A -85,B 0,C 180,E1 23071.118,E2 23071.118} C_VEL
LIN {X 0,Y 473.8,Z 1043.723,A -85,B 0,C 180,E1 23068.353,E2 23068.353} C_VEL
LIN {X 0,Y 473.209,Z 1065.167,A -85,B 0,C 180,E1 23067.753,E2 23067.753} C_VEL
LIN {X 0,Y 472.518,Z 1081.464,A -85,B 0,C 180,E1 23067.062,E2 23067.062} C_VEL
LIN {X 0,Y 471.642,Z 1097.306,A -85,B 0,C 180,E1 23066.166,E2 23066.166} C_VEL
LIN {X 0,Y 470.559,Z 1112.877,A -85,B 0,C 180,E1 23065.015,E2 23065.015} C_VEL
LIN {X 0,Y 469.53,Z 1126.667,A -85,B 0,C 180,E1 23063.734,E2 23063.734} C_VEL
LIN {X 0,Y 468.443,Z 1139.93,A -85,B 0,C 180,E1 23062.198,E2 23062.198} C_VEL
LIN {X 0,Y 467.542,Z 1150.666,A -85,B 0,C 180,E1 23060.663,E2 23060.663} C_VEL
LIN {X 0,Y 466.714,Z 1160.741,A -85,B 0,C 180,E1 23058.875,E2 23058.875} C_VEL
LIN {X 0,Y 466.136,Z 1168.712,A -85,B 0,C 180,E1 23057.09,E2 23057.09} C_VEL
LIN {X 0,Y 465.709,Z 1175.629,A -85,B 0,C 180,E1 23055.058,E2 23055.058} C_VEL
LIN {X 0,Y 465.513,Z 1180.271,A -85,B 0,C 180,E1 23053.161,E2 23053.161} C_VEL
LIN {X 0,Y 465.492,Z 1183.591,A -85,B 0,C 180,E1 23051.007,E2 23051.007} C_VEL
LIN {X 0,Y 465.643,Z 1184.915,A -85,B 0,C 180,E1 23048.986,E2 23048.986} C_VEL
LIN {X 0,Y 466.024,Z 1184.42,A -85,B 0,C 180,E1 23046.777,E2 23046.777} C_VEL
LIN {X 0,Y 466.635,Z 1182.004,A -85,B 0,C 180,E1 23044.671,E2 23044.671} C_VEL
LIN {X 0,Y 467.503,Z 1178.042,A -85,B 0,C 180,E1 23042.697,E2 23042.697} C_VEL
LIN {X 0,Y 468.662,Z 1172.2,A -85,B 0,C 180,E1 23040.733,E2 23040.733} C_VEL
LIN {X 0,Y 470.079,Z 1164.958,A -85,B 0,C 180,E1 23038.903,E2 23038.903} C_VEL
LIN {X 0,Y 471.818,Z 1155.654,A -85,B 0,C 180,E1 23037.085,E2 23037.085} C_VEL
LIN {X 0,Y 473.585,Z 1145.678,A -85,B 0,C 180,E1 23035.52,E2 23035.52} C_VEL
LIN {X 0,Y 475.668,Z 1132.738,A -85,B 0,C 180,E1 23033.906,E2 23033.906} C_VEL
LIN {X 0,Y 477.633,Z 1119.029,A -85,B 0,C 180,E1 23032.542,E2 23032.542} C_VEL
LIN {X 0,Y 479.44,Z 1105.019,A -85,B 0,C 180,E1 23031.424,E2 23031.424} C_VEL
LIN {X 0,Y 481.119,Z 1088.977,A -85,B 0,C 180,E1 23030.429,E2 23030.429} C_VEL
LIN {X 0,Y 482.399,Z 1072.672,A -85,B 0,C 180,E1 23029.671,E2 23029.671} C_VEL
LIN {X 0,Y 485.506,Z 1037.821,A -85,B 0,C 180,E1 23028.42,E2 23028.42} C_VEL
LIN {X 0,Y 493.238,Z 969.488,A -85,B 0,C 180,E1 23026.257,E2 23026.257} C_VEL
LIN {X 0,Y 496.856,Z 933.88,A -85,B 0,C 180,E1 23025.244,E2 23025.244} C_VEL
LIN {X 0,Y 496.97,Z 931.736,A -85,B 0,C 180,E1 23025.076,E2 23025.076} C_VEL
LIN {X 0,Y 504.998,Z 894.531,A -85,B 0,C 180,E1 23021.291,E2 23021.291} C_VEL
LIN {X 0,Y 514.415,Z 859.471,A -85,B 0,C 180,E1 23017.606,E2 23017.606} C_VEL
LIN {X 0,Y 525.664,Z 825.992,A -85,B 0,C 180,E1 23013.935,E2 23013.935} C_VEL
LIN {X 0,Y 535.911,Z 801.443,A -85,B 0,C 180,E1 23011.118,E2 23011.118} C_VEL
LIN {X 0,Y 536.022,Z 796.565,A -85,B 0,C 180,E1 23009.306,E2 23009.306} C_VEL
LIN {X 0,Y 536.441,Z 793.565,A -85,B 0,C 180,E1 23007.533,E2 23007.533} C_VEL
LIN {X 0,Y 537.491,Z 792.122,A -85,B 0,C 180,E1 23005.302,E2 23005.302} C_VEL
LIN {X 0,Y 537.962,Z 794.906,A -85,B 0,C 180,E1 23003.23,E2 23003.23} C_VEL
LIN {X 0,Y 537.936,Z 795.362,A -85,B 0,C 180,E1 23003.056,E2 23003.056} C_VEL
LIN {X 0,Y 525.704,Z 821.94,A -85,B 0,C 180,E1 23000.549,E2 23000.549} C_VEL
LIN {X 0,Y 518.268,Z 843.333,A -85,B 0,C 180,E1 22998.463,E2 22998.463} C_VEL
LIN {X 0,Y 513.427,Z 864.484,A -85,B 0,C 180,E1 22996.259,E2 22996.259} C_VEL
LIN {X 0,Y 511.601,Z 881.938,A -85,B 0,C 180,E1 22994.33,E2 22994.33} C_VEL
LIN {X 0,Y 512.13,Z 899.673,A -85,B 0,C 180,E1 22992.271,E2 22992.271} C_VEL
LIN {X 0,Y 514.95,Z 915.636,A -85,B 0,C 180,E1 22990.348,E2 22990.348} C_VEL
LIN {X 0,Y 520.257,Z 931.651,A -85,B 0,C 180,E1 22988.358,E2 22988.358} C_VEL
LIN {X 0,Y 522.898,Z 938.016,A -85,B 0,C 180,E1 22987.587,E2 22987.587} C_VEL
LIN {X 0,Y 506.225,Z 972.599,A -85,B 0,C 180,E1 22986.196,E2 22986.196} C_VEL
LIN {X 0,Y 496.225,Z 997.979,A -85,B 0,C 180,E1 22984.989,E2 22984.989} C_VEL
LIN {X 0,Y 492.981,Z 1026.926,A -85,B 0,C 180,E1 22984.589,E2 22984.589} C_VEL
LIN {X 0,Y 491.063,Z 1052.408,A -85,B 0,C 180,E1 22983.992,E2 22983.992} C_VEL
LIN {X 0,Y 488.558,Z 1076.224,A -85,B 0,C 180,E1 22983.226,E2 22983.226} C_VEL
LIN {X 0,Y 485.838,Z 1098.979,A -85,B 0,C 180,E1 22982.278,E2 22982.278} C_VEL
LIN {X 0,Y 482.452,Z 1129.218,A -85,B 0,C 180,E1 22980.789,E2 22980.789} C_VEL
LIN {X 0,Y 480.099,Z 1149.331,A -85,B 0,C 180,E1 22979.575,E2 22979.575} C_VEL
LIN {X 0,Y 477.658,Z 1168.783,A -85,B 0,C 180,E1 22978.171,E2 22978.171} C_VEL
LIN {X 0,Y 475.199,Z 1187.364,A -85,B 0,C 180,E1 22976.585,E2 22976.585} C_VEL
LIN {X 0,Y 472.814,Z 1205.062,A -85,B 0,C 180,E1 22974.79,E2 22974.79} C_VEL
LIN {X 0,Y 470.637,Z 1221.161,A -85,B 0,C 180,E1 22972.877,E2 22972.877} C_VEL
LIN {X 0,Y 468.79,Z 1235.701,A -85,B 0,C 180,E1 22970.865,E2 22970.865} C_VEL
LIN {X 0,Y 467.207,Z 1248.896,A -85,B 0,C 180,E1 22968.723,E2 22968.723} C_VEL
LIN {X 0,Y 465.956,Z 1260.834,A -85,B 0,C 180,E1 22966.419,E2 22966.419} C_VEL
LIN {X 0,Y 465.018,Z 1271.596,A -85,B 0,C 180,E1 22963.933,E2 22963.933} C_VEL
LIN {X 0,Y 464.483,Z 1280.095,A -85,B 0,C 180,E1 22961.547,E2 22961.547} C_VEL
LIN {X 0,Y 464.219,Z 1286.767,A -85,B 0,C 180,E1 22959.17,E2 22959.17} C_VEL
LIN {X 0,Y 464.139,Z 1292.114,A -85,B 0,C 180,E1 22956.679,E2 22956.679} C_VEL
LIN {X 0,Y 464.167,Z 1295.667,A -85,B 0,C 180,E1 22954.322,E2 22954.322} C_VEL
LIN {X 0,Y 464.214,Z 1297.747,A -85,B 0,C 180,E1 22951.85,E2 22951.85} C_VEL
LIN {X 0,Y 464.217,Z 1298.319,A -85,B 0,C 180,E1 22949.381,E2 22949.381} C_VEL
LIN {X 0,Y 464.189,Z 1297.292,A -85,B 0,C 180,E1 22947.035,E2 22947.035} C_VEL
LIN {X 0,Y 464.126,Z 1294.543,A -85,B 0,C 180,E1 22944.435,E2 22944.435} C_VEL
LIN {X 0,Y 464.155,Z 1290.307,A -85,B 0,C 180,E1 22941.949,E2 22941.949} C_VEL
LIN {X 0,Y 464.339,Z 1284.31,A -85,B 0,C 180,E1 22939.452,E2 22939.452} C_VEL
LIN {X 0,Y 464.858,Z 1276.155,A -85,B 0,C 180,E1 22936.819,E2 22936.819} C_VEL
LIN {X 0,Y 465.674,Z 1267.013,A -85,B 0,C 180,E1 22934.43,E2 22934.43} C_VEL
LIN {X 0,Y 466.917,Z 1255.874,A -85,B 0,C 180,E1 22932.037,E2 22932.037} C_VEL
LIN {X 0,Y 468.648,Z 1242.658,A -85,B 0,C 180,E1 22929.648,E2 22929.648} C_VEL
LIN {X 0,Y 470.667,Z 1228.825,A -85,B 0,C 180,E1 22927.517,E2 22927.517} C_VEL
LIN {X 0,Y 473.188,Z 1212.684,A -85,B 0,C 180,E1 22925.399,E2 22925.399} C_VEL
LIN {X 0,Y 476.026,Z 1194.937,A -85,B 0,C 180,E1 22923.421,E2 22923.421} C_VEL
LIN {X 0,Y 479.16,Z 1175.582,A -85,B 0,C 180,E1 22921.589,E2 22921.589} C_VEL
LIN {X 0,Y 482.558,Z 1154.494,A -85,B 0,C 180,E1 22919.903,E2 22919.903} C_VEL
LIN {X 0,Y 485.875,Z 1133.355,A -85,B 0,C 180,E1 22918.484,E2 22918.484} C_VEL
LIN {X 0,Y 489.344,Z 1110.435,A -85,B 0,C 180,E1 22917.214,E2 22917.214} C_VEL
LIN {X 0,Y 492.612,Z 1087.342,A -85,B 0,C 180,E1 22916.173,E2 22916.173} C_VEL
LIN {X 0,Y 495.931,Z 1061.91,A -85,B 0,C 180,E1 22915.283,E2 22915.283} C_VEL
LIN {X 0,Y 498.89,Z 1033.365,A -85,B 0,C 180,E1 22914.528,E2 22914.528} C_VEL
LIN {X 0,Y 502.128,Z 1008.247,A -85,B 0,C 180,E1 22914.05,E2 22914.05} C_VEL
LIN {X 0,Y 508.742,Z 970.698,A -85,B 0,C 180,E1 22913.535,E2 22913.535} C_VEL
LIN {X 0,Y 512.908,Z 952.496,A -85,B 0,C 180,E1 22913.377,E2 22913.377} C_VEL
LIN {X 0,Y 521.316,Z 935.927,A -85,B 0,C 180,E1 22912.657,E2 22912.657} C_VEL
LIN {X 0,Y 513.269,Z 918.448,A -85,B 0,C 180,E1 22910.924,E2 22910.924} C_VEL
LIN {X 0,Y 507.302,Z 900.22,A -85,B 0,C 180,E1 22909.189,E2 22909.189} C_VEL
LIN {X 0,Y 505.519,Z 892.386,A -85,B 0,C 180,E1 22908.432,E2 22908.432} C_VEL
LIN {X 0,Y 505.401,Z 881.184,A -85,B 0,C 180,E1 22907.068,E2 22907.068} C_VEL
LIN {X 0,Y 506.901,Z 869.028,A -85,B 0,C 180,E1 22905.763,E2 22905.763} C_VEL
LIN {X 0,Y 509.278,Z 858.042,A -85,B 0,C 180,E1 22904.508,E2 22904.508} C_VEL
LIN {X 0,Y 513.23,Z 845.212,A -85,B 0,C 180,E1 22903.274,E2 22903.274} C_VEL
LIN {X 0,Y 517.573,Z 834.475,A -85,B 0,C 180,E1 22902.131,E2 22902.131} C_VEL
LIN {X 0,Y 523.584,Z 820.887,A -85,B 0,C 180,E1 22901.011,E2 22901.011} C_VEL
LIN {X 0,Y 527.187,Z 814.598,A -85,B 0,C 180,E1 22900.334,E2 22900.334} C_VEL
LIN {X 0,Y 515.391,Z 887.806,A -85,B 0,C 180,E1 22898.434,E2 22898.434} C_VEL
LIN {X 0,Y 506.2,Z 958.674,A -85,B 0,C 180,E1 22896.631,E2 22896.631} C_VEL
LIN {X 0,Y 499.224,Z 1026.749,A -85,B 0,C 180,E1 22894.935,E2 22894.935} C_VEL
LIN {X 0,Y 496.486,Z 1051.175,A -85,B 0,C 180,E1 22894.082,E2 22894.082} C_VEL
LIN {X 0,Y 493.595,Z 1073.454,A -85,B 0,C 180,E1 22893.089,E2 22893.089} C_VEL
LIN {X 0,Y 490.419,Z 1095.442,A -85,B 0,C 180,E1 22891.875,E2 22891.875} C_VEL
LIN {X 0,Y 487.221,Z 1115.646,A -85,B 0,C 180,E1 22890.526,E2 22890.526} C_VEL
LIN {X 0,Y 483.934,Z 1135.087,A -85,B 0,C 180,E1 22888.981,E2 22888.981} C_VEL
LIN {X 0,Y 480.537,Z 1154.214,A -85,B 0,C 180,E1 22887.176,E2 22887.176} C_VEL
LIN {X 0,Y 477.424,Z 1171.121,A -85,B 0,C 180,E1 22885.293,E2 22885.293} C_VEL
LIN {X 0,Y 474.57,Z 1186.554,A -85,B 0,C 180,E1 22883.272,E2 22883.272} C_VEL
LIN {X 0,Y 471.836,Z 1201.245,A -85,B 0,C 180,E1 22880.986,E2 22880.986} C_VEL
LIN {X 0,Y 469.651,Z 1213.274,A -85,B 0,C 180,E1 22878.753,E2 22878.753} C_VEL
LIN {X 0,Y 467.753,Z 1224.508,A -85,B 0,C 180,E1 22876.262,E2 22876.262} C_VEL
LIN {X 0,Y 466.345,Z 1233.765,A -85,B 0,C 180,E1 22873.763,E2 22873.763} C_VEL
LIN {X 0,Y 465.344,Z 1241.494,A -85,B 0,C 180,E1 22871.15,E2 22871.15} C_VEL
LIN {X 0,Y 464.716,Z 1247.04,A -85,B 0,C 180,E1 22868.663,E2 22868.663} C_VEL
LIN {X 0,Y 464.336,Z 1251.393,A -85,B 0,C 180,E1 22865.933,E2 22865.933} C_VEL
LIN {X 0,Y 464.154,Z 1253.891,A -85,B 0,C 180,E1 22863.334,E2 22863.334} C_VEL
LIN {X 0,Y 464.093,Z 1254.68,A -85,B 0,C 180,E1 22860.864,E2 22860.864} C_VEL
LIN {X 0,Y 464.073,Z 1253.938,A -85,B 0,C 180,E1 22858.271,E2 22858.271} C_VEL
LIN {X 0,Y 464.104,Z 1251.783,A -85,B 0,C 180,E1 22855.799,E2 22855.799} C_VEL
LIN {X 0,Y 464.239,Z 1247.98,A -85,B 0,C 180,E1 22853.321,E2 22853.321} C_VEL
LIN {X 0,Y 464.534,Z 1242.343,A -85,B 0,C 180,E1 22850.71,E2 22850.71} C_VEL
LIN {X 0,Y 465.078,Z 1235.289,A -85,B 0,C 180,E1 22848.215,E2 22848.215} C_VEL
LIN {X 0,Y 465.931,Z 1226.308,A -85,B 0,C 180,E1 22845.712,E2 22845.712} C_VEL
LIN {X 0,Y 467.106,Z 1215.89,A -85,B 0,C 180,E1 22843.331,E2 22843.331} C_VEL
LIN {X 0,Y 468.697,Z 1203.431,A -85,B 0,C 180,E1 22840.949,E2 22840.949} C_VEL
LIN {X 0,Y 470.497,Z 1190.292,A -85,B 0,C 180,E1 22838.821,E2 22838.821} C_VEL
LIN {X 0,Y 472.683,Z 1174.757,A -85,B 0,C 180,E1 22836.698,E2 22836.698} C_VEL
LIN {X 0,Y 474.966,Z 1158.719,A -85,B 0,C 180,E1 22834.834,E2 22834.834} C_VEL
LIN {X 0,Y 477.577,Z 1139.969,A -85,B 0,C 180,E1 22832.978,E2 22832.978} C_VEL
LIN {X 0,Y 480.131,Z 1120.832,A -85,B 0,C 180,E1 22831.381,E2 22831.381} C_VEL
LIN {X 0,Y 482.602,Z 1100.851,A -85,B 0,C 180,E1 22829.976,E2 22829.976} C_VEL
LIN {X 0,Y 484.957,Z 1079.852,A -85,B 0,C 180,E1 22828.765,E2 22828.765} C_VEL
LIN {X 0,Y 487.001,Z 1058.644,A -85,B 0,C 180,E1 22827.77,E2 22827.77} C_VEL
LIN {X 0,Y 488.894,Z 1035.169,A -85,B 0,C 180,E1 22826.906,E2 22826.906} C_VEL
LIN {X 0,Y 490.36,Z 1012.464,A -85,B 0,C 180,E1 22826.291,E2 22826.291} C_VEL
LIN {X 0,Y 493.254,Z 942.676,A -85,B 0,C 180,E1 22825.013,E2 22825.013} C_VEL
LIN {X 0,Y 501.921,Z 754.009,A -85,B 0,C 180,E1 22821.588,E2 22821.588} C_VEL
LIN {X 0,Y 500.831,Z 750.703,A -85,B 0,C 180,E1 22821.433,E2 22821.433} C_VEL
LIN {X 0,Y 484.673,Z 719.205,A -85,B 0,C 180,E1 22819.44,E2 22819.44} C_VEL
LIN {X 0,Y 478.416,Z 707.384,A -85,B 0,C 180,E1 22818.619,E2 22818.619} C_VEL
LIN {X 0,Y 471.152,Z 687.679,A -85,B 0,C 180,E1 22815.834,E2 22815.834} C_VEL
LIN {X 0,Y 466.17,Z 674.602,A -85,B 0,C 180,E1 22813.888,E2 22813.888} C_VEL
LIN {X 0,Y 466.167,Z 674.597,A -85,B 0,C 180,E1 22810.214,E2 22810.214} C_VEL
LIN {X 0,Y 466.169,Z 674.595,A -85,B 0,C 180,E1 22806.606,E2 22806.606} C_VEL
LIN {X 0,Y 466.18,Z 674.598,A -85,B 0,C 180,E1 22802.866,E2 22802.866} C_VEL
LIN {X 0,Y 466.177,Z 674.599,A -85,B 0,C 180,E1 22799.195,E2 22799.195} C_VEL
LIN {X 0,Y 466.178,Z 674.6,A -85,B 0,C 180,E1 22795.445,E2 22795.445} C_VEL
LIN {X 0,Y 466.177,Z 674.599,A -85,B 0,C 180,E1 22791.761,E2 22791.761} C_VEL
LIN {X 0,Y 466.175,Z 674.602,A -85,B 0,C 180,E1 22788.121,E2 22788.121} C_VEL
LIN {X 0,Y 466.172,Z 674.594,A -85,B 0,C 180,E1 22784.408,E2 22784.408} C_VEL
LIN {X 0,Y 466.176,Z 674.599,A -85,B 0,C 180,E1 22780.756,E2 22780.756} C_VEL
LIN {X 0,Y 466.168,Z 674.599,A -85,B 0,C 180,E1 22777.024,E2 22777.024} C_VEL
LIN {X 0,Y 466.166,Z 674.594,A -85,B 0,C 180,E1 22773.322,E2 22773.322} C_VEL
LIN {X 0,Y 466.165,Z 674.589,A -85,B 0,C 180,E1 22769.633,E2 22769.633} C_VEL
LIN {X 0,Y 466.167,Z 674.6,A -85,B 0,C 180,E1 22767.534,E2 22767.534} C_VEL
LIN {X 0,Y 465.171,Z 674.729,A -85,B 0,C 180,E1 22766.587,E2 22766.587} C_VEL
LIN {X 0,Y 458.668,Z 675.537,A -85,B 0,C 180,E1 22763.854,E2 22763.854} C_VEL
LIN {X 0,Y 458.23,Z 675.585,A -85,B 0,C 180,E1 22763.228,E2 22763.228} C_VEL
LIN {X 0,Y 458.232,Z 675.582,A -85,B 0,C 180,E1 22759.567,E2 22759.567} C_VEL
LIN {X 0,Y 458.237,Z 675.581,A -85,B 0,C 180,E1 22755.856,E2 22755.856} C_VEL
LIN {X 0,Y 458.231,Z 675.588,A -85,B 0,C 180,E1 22752.061,E2 22752.061} C_VEL
LIN {X 0,Y 458.234,Z 675.59,A -85,B 0,C 180,E1 22748.363,E2 22748.363} C_VEL
LIN {X 0,Y 458.228,Z 675.584,A -85,B 0,C 180,E1 22744.607,E2 22744.607} C_VEL
LIN {X 0,Y 458.241,Z 675.585,A -85,B 0,C 180,E1 22740.886,E2 22740.886} C_VEL
LIN {X 0,Y 458.255,Z 675.775,A -85,B 0,C 180,E1 22737.324,E2 22737.324} C_VEL
LIN {X 0,Y 459.6,Z 679.147,A -85,B 0,C 180,E1 22736.756,E2 22736.756} C_VEL
LIN {X 0,Y 467.491,Z 697.914,A -85,B 0,C 180,E1 22733.671,E2 22733.671} C_VEL
LIN {X 0,Y 474.938,Z 716.98,A -85,B 0,C 180,E1 22730.783,E2 22730.783} C_VEL
LIN {X 0,Y 482.163,Z 737.322,A -85,B 0,C 180,E1 22727.937,E2 22727.937} C_VEL
LIN {X 0,Y 486.827,Z 751.834,A -85,B 0,C 180,E1 22726.038,E2 22726.038} C_VEL
LIN {X 0,Y 482.114,Z 792.273,A -85,B 0,C 180,E1 22722.38,E2 22722.38} C_VEL
LIN {X 0,Y 477.425,Z 836.047,A -85,B 0,C 180,E1 22718.464,E2 22718.464} C_VEL
LIN {X 0,Y 473.173,Z 880.895,A -85,B 0,C 180,E1 22714.495,E2 22714.495} C_VEL
LIN {X 0,Y 470.608,Z 912.16,A -85,B 0,C 180,E1 22711.785,E2 22711.785} C_VEL
LIN {X 0,Y 471.439,Z 923.919,A -85,B 0,C 180,E1 22711.455,E2 22711.455} C_VEL
LIN {X 0,Y 466.306,Z 1038.996,A -85,B 0,C 180,E1 22708.755,E2 22708.755} C_VEL
LIN {X 0,Y 465.551,Z 1064.059,A -85,B 0,C 180,E1 22708.062,E2 22708.062} C_VEL
LIN {X 0,Y 464.848,Z 1080.746,A -85,B 0,C 180,E1 22707.366,E2 22707.366} C_VEL
LIN {X 0,Y 463.91,Z 1097.234,A -85,B 0,C 180,E1 22706.429,E2 22706.429} C_VEL
LIN {X 0,Y 462.845,Z 1112.189,A -85,B 0,C 180,E1 22705.325,E2 22705.325} C_VEL
LIN {X 0,Y 461.732,Z 1126.856,A -85,B 0,C 180,E1 22703.963,E2 22703.963} C_VEL
LIN {X 0,Y 460.64,Z 1139.777,A -85,B 0,C 180,E1 22702.46,E2 22702.46} C_VEL
LIN {X 0,Y 459.704,Z 1150.745,A -85,B 0,C 180,E1 22700.899,E2 22700.899} C_VEL
LIN {X 0,Y 458.833,Z 1160.976,A -85,B 0,C 180,E1 22699.08,E2 22699.08} C_VEL
LIN {X 0,Y 458.226,Z 1169.134,A -85,B 0,C 180,E1 22697.263,E2 22697.263} C_VEL
LIN {X 0,Y 457.776,Z 1176.183,A -85,B 0,C 180,E1 22695.195,E2 22695.195} C_VEL
LIN {X 0,Y 457.56,Z 1181.233,A -85,B 0,C 180,E1 22693.136,E2 22693.136} C_VEL
LIN {X 0,Y 457.545,Z 1184.562,A -85,B 0,C 180,E1 22690.96,E2 22690.96} C_VEL
LIN {X 0,Y 457.713,Z 1185.934,A -85,B 0,C 180,E1 22688.923,E2 22688.923} C_VEL
LIN {X 0,Y 458.133,Z 1185.485,A -85,B 0,C 180,E1 22686.643,E2 22686.643} C_VEL
LIN {X 0,Y 458.795,Z 1183.114,A -85,B 0,C 180,E1 22684.5,E2 22684.5} C_VEL
LIN {X 0,Y 459.723,Z 1179.193,A -85,B 0,C 180,E1 22682.493,E2 22682.493} C_VEL
LIN {X 0,Y 461.05,Z 1173.005,A -85,B 0,C 180,E1 22680.373,E2 22680.373} C_VEL
LIN {X 0,Y 462.585,Z 1165.742,A -85,B 0,C 180,E1 22678.514,E2 22678.514} C_VEL
LIN {X 0,Y 464.587,Z 1155.703,A -85,B 0,C 180,E1 22676.545,E2 22676.545} C_VEL
LIN {X 0,Y 466.472,Z 1145.421,A -85,B 0,C 180,E1 22674.958,E2 22674.958} C_VEL
LIN {X 0,Y 468.557,Z 1133.433,A -85,B 0,C 180,E1 22673.444,E2 22673.444} C_VEL
LIN {X 0,Y 470.647,Z 1119.703,A -85,B 0,C 180,E1 22672.062,E2 22672.062} C_VEL
LIN {X 0,Y 472.543,Z 1105.584,A -85,B 0,C 180,E1 22670.93,E2 22670.93} C_VEL
LIN {X 0,Y 474.343,Z 1089.705,A -85,B 0,C 180,E1 22669.924,E2 22669.924} C_VEL
LIN {X 0,Y 475.835,Z 1072.233,A -85,B 0,C 180,E1 22669.098,E2 22669.098} C_VEL
LIN {X 0,Y 479.356,Z 1036.493,A -85,B 0,C 180,E1 22667.784,E2 22667.784} C_VEL
LIN {X 0,Y 486.591,Z 976.237,A -85,B 0,C 180,E1 22665.819,E2 22665.819} C_VEL
LIN {X 0,Y 491.028,Z 935.655,A -85,B 0,C 180,E1 22664.627,E2 22664.627} C_VEL
LIN {X 0,Y 491.045,Z 933.462,A -85,B 0,C 180,E1 22664.468,E2 22664.468} C_VEL
LIN {X 0,Y 499.933,Z 895.026,A -85,B 0,C 180,E1 22660.488,E2 22660.488} C_VEL
LIN {X 0,Y 509.591,Z 861.439,A -85,B 0,C 180,E1 22656.894,E2 22656.894} C_VEL
LIN {X 0,Y 521.089,Z 829.405,A -85,B 0,C 180,E1 22653.32,E2 22653.32} C_VEL
LIN {X 0,Y 531.056,Z 806.805,A -85,B 0,C 180,E1 22650.69,E2 22650.69} C_VEL
LIN {X 0,Y 531.413,Z 802.353,A -85,B 0,C 180,E1 22648.878,E2 22648.878} C_VEL
LIN {X 0,Y 531.848,Z 799.977,A -85,B 0,C 180,E1 22647.346,E2 22647.346} C_VEL
LIN {X 0,Y 532.956,Z 798.726,A -85,B 0,C 180,E1 22645.256,E2 22645.256} C_VEL
LIN {X 0,Y 533.234,Z 801.118,A -85,B 0,C 180,E1 22643.511,E2 22643.511} C_VEL
LIN {X 0,Y 520.531,Z 827.606,A -85,B 0,C 180,E1 22640.975,E2 22640.975} C_VEL
LIN {X 0,Y 512.748,Z 849.07,A -85,B 0,C 180,E1 22638.823,E2 22638.823} C_VEL
LIN {X 0,Y 507.739,Z 869.726,A -85,B 0,C 180,E1 22636.605,E2 22636.605} C_VEL
LIN {X 0,Y 505.792,Z 887.665,A -85,B 0,C 180,E1 22634.568,E2 22634.568} C_VEL
LIN {X 0,Y 506.218,Z 905.01,A -85,B 0,C 180,E1 22632.492,E2 22632.492} C_VEL
LIN {X 0,Y 509.147,Z 921.559,A -85,B 0,C 180,E1 22630.439,E2 22630.439} C_VEL
LIN {X 0,Y 514.436,Z 937.306,A -85,B 0,C 180,E1 22628.436,E2 22628.436} C_VEL
LIN {X 0,Y 515.587,Z 940.166,A -85,B 0,C 180,E1 22628.073,E2 22628.073} C_VEL
LIN {X 0,Y 499.734,Z 972.94,A -85,B 0,C 180,E1 22626.742,E2 22626.742} C_VEL
LIN {X 0,Y 490.259,Z 996.778,A -85,B 0,C 180,E1 22625.604,E2 22625.604} C_VEL
LIN {X 0,Y 486.767,Z 1026.86,A -85,B 0,C 180,E1 22625.18,E2 22625.18} C_VEL
LIN {X 0,Y 484.646,Z 1052.584,A -85,B 0,C 180,E1 22624.555,E2 22624.555} C_VEL
LIN {X 0,Y 481.914,Z 1076.964,A -85,B 0,C 180,E1 22623.745,E2 22623.745} C_VEL
LIN {X 0,Y 478.918,Z 1100.397,A -85,B 0,C 180,E1 22622.732,E2 22622.732} C_VEL
LIN {X 0,Y 475.622,Z 1124.281,A -85,B 0,C 180,E1 22621.421,E2 22621.421} C_VEL
LIN {X 0,Y 472.766,Z 1147.781,A -85,B 0,C 180,E1 22620.01,E2 22620.01} C_VEL
LIN {X 0,Y 470.231,Z 1167.536,A -85,B 0,C 180,E1 22618.581,E2 22618.581} C_VEL
LIN {X 0,Y 467.58,Z 1186.914,A -85,B 0,C 180,E1 22616.908,E2 22616.908} C_VEL
LIN {X 0,Y 465.157,Z 1204.319,A -85,B 0,C 180,E1 22615.119,E2 22615.119} C_VEL
LIN {X 0,Y 462.869,Z 1220.703,A -85,B 0,C 180,E1 22613.149,E2 22613.149} C_VEL
LIN {X 0,Y 460.954,Z 1235.273,A -85,B 0,C 180,E1 22611.103,E2 22611.103} C_VEL
LIN {X 0,Y 459.317,Z 1248.497,A -85,B 0,C 180,E1 22608.925,E2 22608.925} C_VEL
LIN {X 0,Y 458.023,Z 1260.422,A -85,B 0,C 180,E1 22606.591,E2 22606.591} C_VEL
LIN {X 0,Y 457.048,Z 1271.25,A -85,B 0,C 180,E1 22604.052,E2 22604.052} C_VEL
LIN {X 0,Y 456.496,Z 1279.761,A -85,B 0,C 180,E1 22601.624,E2 22601.624} C_VEL
LIN {X 0,Y 456.225,Z 1286.433,A -85,B 0,C 180,E1 22599.204,E2 22599.204} C_VEL
LIN {X 0,Y 456.147,Z 1291.771,A -85,B 0,C 180,E1 22596.67,E2 22596.67} C_VEL
LIN {X 0,Y 456.18,Z 1295.403,A -85,B 0,C 180,E1 22594.203,E2 22594.203} C_VEL
LIN {X 0,Y 456.227,Z 1297.364,A -85,B 0,C 180,E1 22591.757,E2 22591.757} C_VEL
LIN {X 0,Y 456.23,Z 1297.897,A -85,B 0,C 180,E1 22589.245,E2 22589.245} C_VEL
LIN {X 0,Y 456.19,Z 1296.837,A -85,B 0,C 180,E1 22586.857,E2 22586.857} C_VEL
LIN {X 0,Y 456.128,Z 1294.036,A -85,B 0,C 180,E1 22584.211,E2 22584.211} C_VEL
LIN {X 0,Y 456.169,Z 1289.755,A -85,B 0,C 180,E1 22581.68,E2 22581.68} C_VEL
LIN {X 0,Y 456.379,Z 1283.694,A -85,B 0,C 180,E1 22579.138,E2 22579.138} C_VEL
LIN {X 0,Y 456.927,Z 1275.926,A -85,B 0,C 180,E1 22576.586,E2 22576.586} C_VEL
LIN {X 0,Y 457.869,Z 1266.295,A -85,B 0,C 180,E1 22574.027,E2 22574.027} C_VEL
LIN {X 0,Y 459.225,Z 1255.104,A -85,B 0,C 180,E1 22571.595,E2 22571.595} C_VEL
LIN {X 0,Y 461.109,Z 1241.826,A -85,B 0,C 180,E1 22569.165,E2 22569.165} C_VEL
LIN {X 0,Y 463.288,Z 1227.979,A -85,B 0,C 180,E1 22567.004,E2 22567.004} C_VEL
LIN {X 0,Y 465.983,Z 1211.843,A -85,B 0,C 180,E1 22564.857,E2 22564.857} C_VEL
LIN {X 0,Y 469.024,Z 1194.111,A -85,B 0,C 180,E1 22562.855,E2 22562.855} C_VEL
LIN {X 0,Y 472.243,Z 1175.507,A -85,B 0,C 180,E1 22561.064,E2 22561.064} C_VEL
LIN {X 0,Y 475.843,Z 1154.719,A -85,B 0,C 180,E1 22559.364,E2 22559.364} C_VEL
LIN {X 0,Y 479.501,Z 1132.999,A -85,B 0,C 180,E1 22557.875,E2 22557.875} C_VEL
LIN {X 0,Y 483.177,Z 1110.508,A -85,B 0,C 180,E1 22556.6,E2 22556.6} C_VEL
LIN {X 0,Y 486.821,Z 1086.689,A -85,B 0,C 180,E1 22555.501,E2 22555.501} C_VEL
LIN {X 0,Y 490.464,Z 1060.849,A -85,B 0,C 180,E1 22554.581,E2 22554.581} C_VEL
LIN {X 0,Y 493.682,Z 1032.686,A -85,B 0,C 180,E1 22553.814,E2 22553.814} C_VEL
LIN {X 0,Y 497.451,Z 1005.962,A -85,B 0,C 180,E1 22553.3,E2 22553.3} C_VEL
LIN {X 0,Y 504.183,Z 969.491,A -85,B 0,C 180,E1 22552.799,E2 22552.799} C_VEL
LIN {X 0,Y 510.082,Z 943.598,A -85,B 0,C 180,E1 22552.577,E2 22552.577} C_VEL
LIN {X 0,Y 513.1,Z 937.363,A -85,B 0,C 180,E1 22552.297,E2 22552.297} C_VEL
LIN {X 0,Y 505.671,Z 920.373,A -85,B 0,C 180,E1 22550.573,E2 22550.573} C_VEL
LIN {X 0,Y 503.176,Z 908.701,A -85,B 0,C 180,E1 22549.101,E2 22549.101} C_VEL
LIN {X 0,Y 502.553,Z 896.109,A -85,B 0,C 180,E1 22547.624,E2 22547.624} C_VEL
LIN {X 0,Y 503.245,Z 884.841,A -85,B 0,C 180,E1 22546.255,E2 22546.255} C_VEL
LIN {X 0,Y 505.156,Z 874.252,A -85,B 0,C 180,E1 22545.101,E2 22545.101} C_VEL
LIN {X 0,Y 508.153,Z 863.176,A -85,B 0,C 180,E1 22543.829,E2 22543.829} C_VEL
LIN {X 0,Y 512.701,Z 850.398,A -85,B 0,C 180,E1 22542.589,E2 22542.589} C_VEL
LIN {X 0,Y 517.69,Z 839.478,A -85,B 0,C 180,E1 22541.439,E2 22541.439} C_VEL
LIN {X 0,Y 521.568,Z 831.577,A -85,B 0,C 180,E1 22540.733,E2 22540.733} C_VEL
LIN {X 0,Y 509.361,Z 903.973,A -85,B 0,C 180,E1 22538.816,E2 22538.816} C_VEL
LIN {X 0,Y 499.962,Z 972.903,A -85,B 0,C 180,E1 22537.03,E2 22537.03} C_VEL
LIN {X 0,Y 493.849,Z 1027.809,A -85,B 0,C 180,E1 22535.607,E2 22535.607} C_VEL
LIN {X 0,Y 490.971,Z 1051.328,A -85,B 0,C 180,E1 22534.767,E2 22534.767} C_VEL
LIN {X 0,Y 487.641,Z 1074.986,A -85,B 0,C 180,E1 22533.687,E2 22533.687} C_VEL
LIN {X 0,Y 484.126,Z 1097.45,A -85,B 0,C 180,E1 22532.409,E2 22532.409} C_VEL
LIN {X 0,Y 480.655,Z 1117.775,A -85,B 0,C 180,E1 22531.009,E2 22531.009} C_VEL
LIN {X 0,Y 477.152,Z 1137.016,A -85,B 0,C 180,E1 22529.433,E2 22529.433} C_VEL
LIN {X 0,Y 473.685,Z 1155.22,A -85,B 0,C 180,E1 22527.671,E2 22527.671} C_VEL
LIN {X 0,Y 470.431,Z 1171.788,A -85,B 0,C 180,E1 22525.789,E2 22525.789} C_VEL
LIN {X 0,Y 467.359,Z 1187.317,A -85,B 0,C 180,E1 22523.717,E2 22523.717} C_VEL
LIN {X 0,Y 464.526,Z 1201.541,A -85,B 0,C 180,E1 22521.465,E2 22521.465} C_VEL
LIN {X 0,Y 462.184,Z 1213.578,A -85,B 0,C 180,E1 22519.198,E2 22519.198} C_VEL
LIN {X 0,Y 460.139,Z 1224.826,A -85,B 0,C 180,E1 22516.669,E2 22516.669} C_VEL
LIN {X 0,Y 458.613,Z 1234.085,A -85,B 0,C 180,E1 22514.134,E2 22514.134} C_VEL
LIN {X 0,Y 457.506,Z 1241.837,A -85,B 0,C 180,E1 22511.472,E2 22511.472} C_VEL
LIN {X 0,Y 456.785,Z 1247.654,A -85,B 0,C 180,E1 22508.814,E2 22508.814} C_VEL
LIN {X 0,Y 456.386,Z 1251.78,A -85,B 0,C 180,E1 22506.163,E2 22506.163} C_VEL
LIN {X 0,Y 456.18,Z 1254.3,A -85,B 0,C 180,E1 22503.519,E2 22503.519} C_VEL
LIN {X 0,Y 456.104,Z 1255.09,A -85,B 0,C 180,E1 22501.005,E2 22501.005} C_VEL
LIN {X 0,Y 456.079,Z 1254.361,A -85,B 0,C 180,E1 22498.367,E2 22498.367} C_VEL
LIN {X 0,Y 456.11,Z 1252.204,A -85,B 0,C 180,E1 22495.851,E2 22495.851} C_VEL
LIN {X 0,Y 456.246,Z 1248.399,A -85,B 0,C 180,E1 22493.33,E2 22493.33} C_VEL
LIN {X 0,Y 456.55,Z 1242.753,A -85,B 0,C 180,E1 22490.673,E2 22490.673} C_VEL
LIN {X 0,Y 457.112,Z 1235.681,A -85,B 0,C 180,E1 22488.134,E2 22488.134} C_VEL
LIN {X 0,Y 457.993,Z 1226.674,A -85,B 0,C 180,E1 22485.588,E2 22485.588} C_VEL
LIN {X 0,Y 459.209,Z 1216.225,A -85,B 0,C 180,E1 22483.166,E2 22483.166} C_VEL
LIN {X 0,Y 460.898,Z 1203.387,A -85,B 0,C 180,E1 22480.686,E2 22480.686} C_VEL
LIN {X 0,Y 462.838,Z 1189.66,A -85,B 0,C 180,E1 22478.453,E2 22478.453} C_VEL
LIN {X 0,Y 465.13,Z 1174,A -85,B 0,C 180,E1 22476.297,E2 22476.297} C_VEL
LIN {X 0,Y 467.586,Z 1157.157,A -85,B 0,C 180,E1 22474.34,E2 22474.34} C_VEL
LIN {X 0,Y 470.145,Z 1139.289,A -85,B 0,C 180,E1 22472.574,E2 22472.574} C_VEL
LIN {X 0,Y 472.871,Z 1119.233,A -85,B 0,C 180,E1 22470.9,E2 22470.9} C_VEL
LIN {X 0,Y 475.327,Z 1099.815,A -85,B 0,C 180,E1 22469.538,E2 22469.538} C_VEL
LIN {X 0,Y 477.765,Z 1078.662,A -85,B 0,C 180,E1 22468.311,E2 22468.311} C_VEL
LIN {X 0,Y 479.871,Z 1057.082,A -85,B 0,C 180,E1 22467.303,E2 22467.303} C_VEL
LIN {X 0,Y 481.723,Z 1034.575,A -85,B 0,C 180,E1 22466.478,E2 22466.478} C_VEL
LIN {X 0,Y 483.262,Z 1010.836,A -85,B 0,C 180,E1 22465.839,E2 22465.839} C_VEL
LIN {X 0,Y 495.224,Z 755.834,A -85,B 0,C 180,E1 22461.123,E2 22461.123} C_VEL
LIN {X 0,Y 479.346,Z 724.617,A -85,B 0,C 180,E1 22459.128,E2 22459.128} C_VEL
LIN {X 0,Y 470.267,Z 707.602,A -85,B 0,C 180,E1 22457.908,E2 22457.908} C_VEL
LIN {X 0,Y 462.9,Z 687.879,A -85,B 0,C 180,E1 22455.062,E2 22455.062} C_VEL
LIN {X 0,Y 458.239,Z 675.589,A -85,B 0,C 180,E1 22453.214,E2 22453.214} C_VEL
LIN {X 0,Y 458.237,Z 675.586,A -85,B 0,C 180,E1 22449.419,E2 22449.419} C_VEL
LIN {X 0,Y 458.24,Z 675.592,A -85,B 0,C 180,E1 22445.736,E2 22445.736} C_VEL
LIN {X 0,Y 458.228,Z 675.587,A -85,B 0,C 180,E1 22441.915,E2 22441.915} C_VEL
LIN {X 0,Y 458.237,Z 675.585,A -85,B 0,C 180,E1 22438.263,E2 22438.263} C_VEL
LIN {X 0,Y 458.227,Z 675.589,A -85,B 0,C 180,E1 22434.495,E2 22434.495} C_VEL
LIN {X 0,Y 458.238,Z 675.587,A -85,B 0,C 180,E1 22430.836,E2 22430.836} C_VEL
LIN {X 0,Y 458.227,Z 675.588,A -85,B 0,C 180,E1 22427.107,E2 22427.107} C_VEL
LIN {X 0,Y 458.234,Z 675.577,A -85,B 0,C 180,E1 22423.375,E2 22423.375} C_VEL
LIN {X 0,Y 458.228,Z 675.586,A -85,B 0,C 180,E1 22419.674,E2 22419.674} C_VEL
LIN {X 0,Y 458.243,Z 675.589,A -85,B 0,C 180,E1 22416.014,E2 22416.014} C_VEL
LIN {X 0,Y 458.232,Z 675.59,A -85,B 0,C 180,E1 22412.253,E2 22412.253} C_VEL
LIN {X 0,Y 458.242,Z 675.584,A -85,B 0,C 180,E1 22408.626,E2 22408.626} C_VEL
LIN {X 0,Y 458.237,Z 675.585,A -85,B 0,C 180,E1 22404.869,E2 22404.869} C_VEL
LIN {X 0,Y 458.23,Z 675.585,A -85,B 0,C 180,E1 22403.228,E2 22403.228} C_VEL
LIN {X 0,Y 457.236,Z 675.706,A -85,B 0,C 180,E1 22402.265,E2 22402.265} C_VEL
LIN {X 0,Y 450.718,Z 676.519,A -85,B 0,C 180,E1 22399.484,E2 22399.484} C_VEL
LIN {X 0,Y 450.288,Z 676.568,A -85,B 0,C 180,E1 22398.847,E2 22398.847} C_VEL
LIN {X 0,Y 450.291,Z 676.573,A -85,B 0,C 180,E1 22395.075,E2 22395.075} C_VEL
LIN {X 0,Y 450.298,Z 676.579,A -85,B 0,C 180,E1 22391.354,E2 22391.354} C_VEL
LIN {X 0,Y 450.288,Z 676.576,A -85,B 0,C 180,E1 22387.686,E2 22387.686} C_VEL
LIN {X 0,Y 450.298,Z 676.578,A -85,B 0,C 180,E1 22383.92,E2 22383.92} C_VEL
LIN {X 0,Y 450.303,Z 676.574,A -85,B 0,C 180,E1 22380.175,E2 22380.175} C_VEL
LIN {X 0,Y 450.296,Z 676.588,A -85,B 0,C 180,E1 22378.212,E2 22378.212} C_VEL
LIN {X 0,Y 451.652,Z 680.118,A -85,B 0,C 180,E1 22377.608,E2 22377.608} C_VEL
LIN {X 0,Y 459.551,Z 698.663,A -85,B 0,C 180,E1 22374.464,E2 22374.464} C_VEL
LIN {X 0,Y 467.103,Z 717.899,A -85,B 0,C 180,E1 22371.473,E2 22371.473} C_VEL
LIN {X 0,Y 474.37,Z 738.208,A -85,B 0,C 180,E1 22368.561,E2 22368.561} C_VEL
LIN {X 0,Y 479.698,Z 755.012,A -85,B 0,C 180,E1 22366.327,E2 22366.327} C_VEL
LIN {X 0,Y 474.891,Z 794.872,A -85,B 0,C 180,E1 22362.686,E2 22362.686} C_VEL
LIN {X 0,Y 470.116,Z 838.068,A -85,B 0,C 180,E1 22358.783,E2 22358.783} C_VEL
LIN {X 0,Y 465.708,Z 882.971,A -85,B 0,C 180,E1 22354.764,E2 22354.764} C_VEL
LIN {X 0,Y 463.156,Z 912.893,A -85,B 0,C 180,E1 22352.138,E2 22352.138} C_VEL
LIN {X 0,Y 463.975,Z 924.718,A -85,B 0,C 180,E1 22351.802,E2 22351.802} C_VEL
LIN {X 0,Y 459.009,Z 1030.23,A -85,B 0,C 180,E1 22349.265,E2 22349.265} C_VEL
LIN {X 0,Y 457.872,Z 1063.458,A -85,B 0,C 180,E1 22348.356,E2 22348.356} C_VEL
LIN {X 0,Y 457.159,Z 1080.418,A -85,B 0,C 180,E1 22347.654,E2 22347.654} C_VEL
LIN {X 0,Y 456.185,Z 1097.105,A -85,B 0,C 180,E1 22346.701,E2 22346.701} C_VEL
LIN {X 0,Y 455.087,Z 1112.281,A -85,B 0,C 180,E1 22345.578,E2 22345.578} C_VEL
LIN {X 0,Y 453.927,Z 1127.138,A -85,B 0,C 180,E1 22344.187,E2 22344.187} C_VEL
LIN {X 0,Y 452.848,Z 1139.623,A -85,B 0,C 180,E1 22342.731,E2 22342.731} C_VEL
LIN {X 0,Y 451.796,Z 1151.617,A -85,B 0,C 180,E1 22341.01,E2 22341.01} C_VEL
LIN {X 0,Y 450.902,Z 1161.878,A -85,B 0,C 180,E1 22339.157,E2 22339.157} C_VEL
LIN {X 0,Y 450.276,Z 1170.131,A -85,B 0,C 180,E1 22337.289,E2 22337.289} C_VEL
LIN {X 0,Y 449.82,Z 1177.108,A -85,B 0,C 180,E1 22335.207,E2 22335.207} C_VEL
LIN {X 0,Y 449.605,Z 1182.182,A -85,B 0,C 180,E1 22333.111,E2 22333.111} C_VEL
LIN {X 0,Y 449.598,Z 1185.54,A -85,B 0,C 180,E1 22330.897,E2 22330.897} C_VEL
LIN {X 0,Y 449.79,Z 1186.958,A -85,B 0,C 180,E1 22328.823,E2 22328.823} C_VEL
LIN {X 0,Y 450.242,Z 1186.551,A -85,B 0,C 180,E1 22326.503,E2 22326.503} C_VEL
LIN {X 0,Y 450.96,Z 1184.229,A -85,B 0,C 180,E1 22324.323,E2 22324.323} C_VEL
LIN {X 0,Y 452.029,Z 1180.082,A -85,B 0,C 180,E1 22322.155,E2 22322.155} C_VEL
LIN {X 0,Y 453.471,Z 1173.865,A -85,B 0,C 180,E1 22320,E2 22320} C_VEL
LIN {X 0,Y 455.114,Z 1166.514,A -85,B 0,C 180,E1 22318.111,E2 22318.111} C_VEL
LIN {X 0,Y 457.26,Z 1156.459,A -85,B 0,C 180,E1 22316.113,E2 22316.113} C_VEL
LIN {X 0,Y 459.454,Z 1145.334,A -85,B 0,C 180,E1 22314.38,E2 22314.38} C_VEL
LIN {X 0,Y 461.577,Z 1133.596,A -85,B 0,C 180,E1 22312.907,E2 22312.907} C_VEL
LIN {X 0,Y 463.813,Z 1119.784,A -85,B 0,C 180,E1 22311.508,E2 22311.508} C_VEL
LIN {X 0,Y 465.954,Z 1104.734,A -85,B 0,C 180,E1 22310.302,E2 22310.302} C_VEL
LIN {X 0,Y 467.631,Z 1090.595,A -85,B 0,C 180,E1 22309.404,E2 22309.404} C_VEL
LIN {X 0,Y 469.209,Z 1073.252,A -85,B 0,C 180,E1 22308.569,E2 22308.569} C_VEL
LIN {X 0,Y 473.04,Z 1037.694,A -85,B 0,C 180,E1 22307.208,E2 22307.208} C_VEL
LIN {X 0,Y 480.803,Z 977.008,A -85,B 0,C 180,E1 22305.172,E2 22305.172} C_VEL
LIN {X 0,Y 485.3,Z 937.551,A -85,B 0,C 180,E1 22303.996,E2 22303.996} C_VEL
LIN {X 0,Y 485.244,Z 935.382,A -85,B 0,C 180,E1 22303.848,E2 22303.848} C_VEL
LIN {X 0,Y 493.898,Z 899.884,A -85,B 0,C 180,E1 22300.116,E2 22300.116} C_VEL
LIN {X 0,Y 504.293,Z 865.576,A -85,B 0,C 180,E1 22296.389,E2 22296.389} C_VEL
LIN {X 0,Y 515.905,Z 834.797,A -85,B 0,C 180,E1 22292.905,E2 22292.905} C_VEL
LIN {X 0,Y 526.338,Z 812.239,A -85,B 0,C 180,E1 22290.242,E2 22290.242} C_VEL
LIN {X 0,Y 526.853,Z 808.063,A -85,B 0,C 180,E1 22288.412,E2 22288.412} C_VEL
LIN {X 0,Y 527.337,Z 806.318,A -85,B 0,C 180,E1 22287.031,E2 22287.031} C_VEL
LIN {X 0,Y 528.401,Z 805.308,A -85,B 0,C 180,E1 22285.279,E2 22285.279} C_VEL
LIN {X 0,Y 528.414,Z 807.123,A -85,B 0,C 180,E1 22283.95,E2 22283.95} C_VEL
LIN {X 0,Y 515.689,Z 832.61,A -85,B 0,C 180,E1 22281.474,E2 22281.474} C_VEL
LIN {X 0,Y 507.829,Z 853.083,A -85,B 0,C 180,E1 22279.375,E2 22279.375} C_VEL
LIN {X 0,Y 502.429,Z 873.772,A -85,B 0,C 180,E1 22277.108,E2 22277.108} C_VEL
LIN {X 0,Y 500.094,Z 891.348,A -85,B 0,C 180,E1 22275.052,E2 22275.052} C_VEL
LIN {X 0,Y 500.249,Z 908.91,A -85,B 0,C 180,E1 22272.907,E2 22272.907} C_VEL
LIN {X 0,Y 502.736,Z 924.912,A -85,B 0,C 180,E1 22270.867,E2 22270.867} C_VEL
LIN {X 0,Y 508.024,Z 941.518,A -85,B 0,C 180,E1 22268.703,E2 22268.703} C_VEL
LIN {X 0,Y 508.319,Z 942.642,A -85,B 0,C 180,E1 22268.573,E2 22268.573} C_VEL
LIN {X 0,Y 494.038,Z 971.938,A -85,B 0,C 180,E1 22267.383,E2 22267.383} C_VEL
LIN {X 0,Y 484.454,Z 995.478,A -85,B 0,C 180,E1 22266.248,E2 22266.248} C_VEL
LIN {X 0,Y 480.67,Z 1026.804,A -85,B 0,C 180,E1 22265.795,E2 22265.795} C_VEL
LIN {X 0,Y 478.501,Z 1051.352,A -85,B 0,C 180,E1 22265.187,E2 22265.187} C_VEL
LIN {X 0,Y 475.518,Z 1076.394,A -85,B 0,C 180,E1 22264.334,E2 22264.334} C_VEL
LIN {X 0,Y 472.371,Z 1099.587,A -85,B 0,C 180,E1 22263.316,E2 22263.316} C_VEL
LIN {X 0,Y 469.049,Z 1122.244,A -85,B 0,C 180,E1 22262.057,E2 22262.057} C_VEL
LIN {X 0,Y 464.039,Z 1156.91,A -85,B 0,C 180,E1 22259.706,E2 22259.706} C_VEL
LIN {X 0,Y 461.453,Z 1175.978,A -85,B 0,C 180,E1 22258.186,E2 22258.186} C_VEL
LIN {X 0,Y 458.84,Z 1194.156,A -85,B 0,C 180,E1 22256.462,E2 22256.462} C_VEL
LIN {X 0,Y 456.443,Z 1210.948,A -85,B 0,C 180,E1 22254.594,E2 22254.594} C_VEL
LIN {X 0,Y 454.196,Z 1226.877,A -85,B 0,C 180,E1 22252.521,E2 22252.521} C_VEL
LIN {X 0,Y 452.27,Z 1241.356,A -85,B 0,C 180,E1 22250.308,E2 22250.308} C_VEL
LIN {X 0,Y 450.716,Z 1254.249,A -85,B 0,C 180,E1 22247.959,E2 22247.959} C_VEL
LIN {X 0,Y 449.574,Z 1265.132,A -85,B 0,C 180,E1 22245.609,E2 22245.609} C_VEL
LIN {X 0,Y 448.808,Z 1274.719,A -85,B 0,C 180,E1 22243.133,E2 22243.133} C_VEL
LIN {X 0,Y 448.356,Z 1282.406,A -85,B 0,C 180,E1 22240.665,E2 22240.665} C_VEL
LIN {X 0,Y 448.183,Z 1288.695,A -85,B 0,C 180,E1 22238.078,E2 22238.078} C_VEL
LIN {X 0,Y 448.167,Z 1293.133,A -85,B 0,C 180,E1 22235.632,E2 22235.632} C_VEL
LIN {X 0,Y 448.214,Z 1295.926,A -85,B 0,C 180,E1 22233.195,E2 22233.195} C_VEL
LIN {X 0,Y 448.244,Z 1297.384,A -85,B 0,C 180,E1 22230.637,E2 22230.637} C_VEL
LIN {X 0,Y 448.225,Z 1297.221,A -85,B 0,C 180,E1 22228.209,E2 22228.209} C_VEL
LIN {X 0,Y 448.157,Z 1295.376,A -85,B 0,C 180,E1 22225.52,E2 22225.52} C_VEL
LIN {X 0,Y 448.13,Z 1292.039,A -85,B 0,C 180,E1 22222.949,E2 22222.949} C_VEL
LIN {X 0,Y 448.246,Z 1286.945,A -85,B 0,C 180,E1 22220.368,E2 22220.368} C_VEL
LIN {X 0,Y 448.667,Z 1279.815,A -85,B 0,C 180,E1 22217.645,E2 22217.645} C_VEL
LIN {X 0,Y 449.448,Z 1271.203,A -85,B 0,C 180,E1 22215.043,E2 22215.043} C_VEL
LIN {X 0,Y 450.722,Z 1260.536,A -85,B 0,C 180,E1 22212.438,E2 22212.438} C_VEL
LIN {X 0,Y 452.459,Z 1248.382,A -85,B 0,C 180,E1 22209.967,E2 22209.967} C_VEL
LIN {X 0,Y 454.777,Z 1234.016,A -85,B 0,C 180,E1 22207.506,E2 22207.506} C_VEL
LIN {X 0,Y 457.507,Z 1218.516,A -85,B 0,C 180,E1 22205.257,E2 22205.257} C_VEL
LIN {X 0,Y 460.694,Z 1201.044,A -85,B 0,C 180,E1 22203.1,E2 22203.1} C_VEL
LIN {X 0,Y 464.179,Z 1182.321,A -85,B 0,C 180,E1 22201.149,E2 22201.149} C_VEL
LIN {X 0,Y 467.776,Z 1162.837,A -85,B 0,C 180,E1 22199.419,E2 22199.419} C_VEL
LIN {X 0,Y 471.778,Z 1141.047,A -85,B 0,C 180,E1 22197.788,E2 22197.788} C_VEL
LIN {X 0,Y 475.813,Z 1118.307,A -85,B 0,C 180,E1 22196.376,E2 22196.376} C_VEL
LIN {X 0,Y 479.813,Z 1094.736,A -85,B 0,C 180,E1 22195.179,E2 22195.179} C_VEL
LIN {X 0,Y 483.581,Z 1071.048,A -85,B 0,C 180,E1 22194.221,E2 22194.221} C_VEL
LIN {X 0,Y 487.2,Z 1045.219,A -85,B 0,C 180,E1 22193.41,E2 22193.41} C_VEL
LIN {X 0,Y 490.239,Z 1021.33,A -85,B 0,C 180,E1 22192.834,E2 22192.834} C_VEL
LIN {X 0,Y 495.076,Z 993.106,A -85,B 0,C 180,E1 22192.362,E2 22192.362} C_VEL
LIN {X 0,Y 500.246,Z 967.017,A -85,B 0,C 180,E1 22192.022,E2 22192.022} C_VEL
LIN {X 0,Y 506.215,Z 940.136,A -85,B 0,C 180,E1 22191.779,E2 22191.779} C_VEL
LIN {X 0,Y 501.977,Z 925.693,A -85,B 0,C 180,E1 22190.031,E2 22190.031} C_VEL
LIN {X 0,Y 500.033,Z 914.177,A -85,B 0,C 180,E1 22188.54,E2 22188.54} C_VEL
LIN {X 0,Y 499.938,Z 901.505,A -85,B 0,C 180,E1 22187.016,E2 22187.016} C_VEL
LIN {X 0,Y 501.262,Z 890.042,A -85,B 0,C 180,E1 22185.599,E2 22185.599} C_VEL
LIN {X 0,Y 503.692,Z 879.485,A -85,B 0,C 180,E1 22184.429,E2 22184.429} C_VEL
LIN {X 0,Y 507.397,Z 868.196,A -85,B 0,C 180,E1 22183.13,E2 22183.13} C_VEL
LIN {X 0,Y 512.458,Z 855.692,A -85,B 0,C 180,E1 22181.915,E2 22181.915} C_VEL
LIN {X 0,Y 515.988,Z 848.814,A -85,B 0,C 180,E1 22181.135,E2 22181.135} C_VEL
LIN {X 0,Y 503.327,Z 920.603,A -85,B 0,C 180,E1 22179.201,E2 22179.201} C_VEL
LIN {X 0,Y 493.744,Z 987.512,A -85,B 0,C 180,E1 22177.432,E2 22177.432} C_VEL
LIN {X 0,Y 488.713,Z 1029.089,A -85,B 0,C 180,E1 22176.307,E2 22176.307} C_VEL
LIN {X 0,Y 485.516,Z 1052.802,A -85,B 0,C 180,E1 22175.432,E2 22175.432} C_VEL
LIN {X 0,Y 481.98,Z 1075.803,A -85,B 0,C 180,E1 22174.352,E2 22174.352} C_VEL
LIN {X 0,Y 478.07,Z 1098.925,A -85,B 0,C 180,E1 22173.007,E2 22173.007} C_VEL
LIN {X 0,Y 474.226,Z 1119.822,A -85,B 0,C 180,E1 22171.527,E2 22171.527} C_VEL
LIN {X 0,Y 470.31,Z 1139.827,A -85,B 0,C 180,E1 22169.834,E2 22169.834} C_VEL
LIN {X 0,Y 466.67,Z 1157.554,A -85,B 0,C 180,E1 22168.054,E2 22168.054} C_VEL
LIN {X 0,Y 463.145,Z 1174.24,A -85,B 0,C 180,E1 22166.088,E2 22166.088} C_VEL
LIN {X 0,Y 459.926,Z 1189.396,A -85,B 0,C 180,E1 22163.988,E2 22163.988} C_VEL
LIN {X 0,Y 456.973,Z 1203.396,A -85,B 0,C 180,E1 22161.702,E2 22161.702} C_VEL
LIN {X 0,Y 454.387,Z 1215.888,A -85,B 0,C 180,E1 22159.259,E2 22159.259} C_VEL
LIN {X 0,Y 452.366,Z 1226.205,A -85,B 0,C 180,E1 22156.832,E2 22156.832} C_VEL
LIN {X 0,Y 450.686,Z 1235.65,A -85,B 0,C 180,E1 22154.126,E2 22154.126} C_VEL
LIN {X 0,Y 449.592,Z 1242.848,A -85,B 0,C 180,E1 22151.546,E2 22151.546} C_VEL
LIN {X 0,Y 448.835,Z 1248.536,A -85,B 0,C 180,E1 22148.842,E2 22148.842} C_VEL
LIN {X 0,Y 448.41,Z 1252.484,A -85,B 0,C 180,E1 22146.144,E2 22146.144} C_VEL
LIN {X 0,Y 448.191,Z 1254.833,A -85,B 0,C 180,E1 22143.453,E2 22143.453} C_VEL
LIN {X 0,Y 448.116,Z 1255.529,A -85,B 0,C 180,E1 22140.895,E2 22140.895} C_VEL
LIN {X 0,Y 448.088,Z 1254.703,A -85,B 0,C 180,E1 22138.338,E2 22138.338} C_VEL
LIN {X 0,Y 448.119,Z 1252.463,A -85,B 0,C 180,E1 22135.777,E2 22135.777} C_VEL
LIN {X 0,Y 448.265,Z 1248.586,A -85,B 0,C 180,E1 22133.211,E2 22133.211} C_VEL
